           "LBP_AlarmMsgs".UserA[05].A70UUxx[00] := FALSE;

           "LBP_AlarmMsgs".UserA[06].A70UUxx[00] := FALSE;
           "LBP_AlarmMsgs".UserA[06].A70UUxx[01] := FALSE;
           "LBP_AlarmMsgs".UserA[06].A70UUxx[02] := FALSE;
           "LBP_AlarmMsgs".UserA[06].A70UUxx[03] := FALSE;
           "LBP_AlarmMsgs".UserA[06].A70UUxx[23] := FALSE;
           "LBP_AlarmMsgs".UserA[06].A70UUxx[25] := FALSE;
       END_IF;
   END_REGION

   REGION Ack alarm level 6
       IF "MCP1_In".reset THEN
           "LBP_AlarmMsgs".UserA[04].A70UUxx[02] := FALSE;
       END_IF;
   END_REGION

   REGION Ack alarm RID 5102xx
       IF "LBP_Chan1".E_ChanReset THEN
           "LBP_AlarmMsgs".ChanA[1].RID_5C02xx[00] := FALSE;
           "LBP_AlarmMsgs".ChanA[1].RID_5C02xx[01] := FALSE;
           "LBP_AlarmMsgs".ChanA[1].RID_5C02xx[02] := FALSE;
           "LBP_AlarmMsgs".ChanA[1].RID_5C02xx[03] := FALSE;
           "LBP_AlarmMsgs".ChanA[1].RID_5C02xx[04] := FALSE;
           "LBP_AlarmMsgs".ChanA[1].RID_5C02xx[05] := FALSE;
           "LBP_AlarmMsgs".ChanA[1].RID_5C02xx[06] := FALSE;
           "LBP_AlarmMsgs".ChanA[1].RID_5C02xx[07] := FALSE;
           "LBP_AlarmMsgs".ChanA[1].RID_5C02xx[08] := FALSE;
           "LBP_AlarmMsgs".ChanA[1].RID_5C02xx[09] := FALSE;
           "LBP_AlarmMsgs".ChanA[1].RID_5C02xx[10] := FALSE;
           "LBP_AlarmMsgs".ChanA[1].RID_5C02xx[11] := FALSE;
           "LBP_AlarmMsgs".ChanA[1].RID_5C02xx[12] := FALSE;
           "LBP_AlarmMsgs".ChanA[1].RID_5C02xx[13] := FALSE;
           "LBP_AlarmMsgs".ChanA[1].RID_5C02xx[14] := FALSE;
           "LBP_AlarmMsgs".ChanA[1].RID_5C02xx[15] := FALSE;
       END_IF;
   END_REGION
END_FUNCTION_BLOCK

FUNCTION_BLOCK "FB_Msg"   // FB84, SCL
{ S7_Optimized_Access := 'TRUE' }
// stored: MemoryReserve 100, SetENOAutomatically false
   VAR
      sSeverity : Byte;
      sMemoNumberOfActiveAlarms : DInt;
      sTON_On : TON_TIME;
      sTON_OFF { S7_SetPoint := 'True'} : TON_TIME;
      sPulseUpdateAlarms { S7_SetPoint := 'True'} : Bool;
      sRT_PulseUpdateAlarms : R_TRIG;
   END_VAR
   VAR_TEMP
      tIndex1 : Int;
      tIndex2 : Int;
      tResultByte0 : Int;
   END_VAR
   VAR CONSTANT
      MSG_SIZE : Int := 95;
   END_VAR
BEGIN
   // REGION Test
   //     FOR #tIndex := 0 TO #MSG_SIZE DO
   //         #tResultByte0 := PEEK(area := 16#84, dbNumber := 2, byteOffset := #tIndex + 554);
   //         "Db_Messages".Msg[#tIndex].ID := #tIndex;
   //         "Db_Messages".Msg[#tIndex].Number := INT_TO_DINT(#tIndex) + 70000;
   //         "Db_Messages".Msg[#tIndex].Active := #tResultByte0.%X0;
   //     END_FOR;
   // END_REGION

   REGION Format Msg
       // Mise en forme des alarmes (DB2) dans DB_FormatMsg
       FOR #tIndex1 := 0 TO 8 DO
           FOR #tIndex2 := 0 TO 7 DO
               #tResultByte0 := PEEK(area := 16#84, dbNumber := 2, byteOffset := #tIndex2 + 554 + (#tIndex1 * 8));
               "DB_FormatMsg".Msg[(#tIndex2 * 8) + (#tIndex1 * 64) + 0].Id := INT_TO_DINT((#tIndex2 * 8) + 0) + 70000 + (#tIndex1 * 100);
               "DB_FormatMsg".Msg[(#tIndex2 * 8) + (#tIndex1 * 64) + 1].Id := INT_TO_DINT((#tIndex2 * 8) + 1) + 70000 + (#tIndex1 * 100);
               "DB_FormatMsg".Msg[(#tIndex2 * 8) + (#tIndex1 * 64) + 2].Id := INT_TO_DINT((#tIndex2 * 8) + 2) + 70000 + (#tIndex1 * 100);
               "DB_FormatMsg".Msg[(#tIndex2 * 8) + (#tIndex1 * 64) + 3].Id := INT_TO_DINT((#tIndex2 * 8) + 3) + 70000 + (#tIndex1 * 100);
               "DB_FormatMsg".Msg[(#tIndex2 * 8) + (#tIndex1 * 64) + 4].Id := INT_TO_DINT((#tIndex2 * 8) + 4) + 70000 + (#tIndex1 * 100);
               "DB_FormatMsg".Msg[(#tIndex2 * 8) + (#tIndex1 * 64) + 5].Id := INT_TO_DINT((#tIndex2 * 8) + 5) + 70000 + (#tIndex1 * 100);
               "DB_FormatMsg".Msg[(#tIndex2 * 8) + (#tIndex1 * 64) + 6].Id := INT_TO_DINT((#tIndex2 * 8) + 6) + 70000 + (#tIndex1 * 100);
               "DB_FormatMsg".Msg[(#tIndex2 * 8) + (#tIndex1 * 64) + 7].Id := INT_TO_DINT((#tIndex2 * 8) + 7) + 70000 + (#tIndex1 * 100);

               "DB_FormatMsg".Msg[(#tIndex2 * 8) + (#tIndex1 * 64) + 0].Active := #tResultByte0.%X0;
               "DB_FormatMsg".Msg[(#tIndex2 * 8) + (#tIndex1 * 64) + 1].Active := #tResultByte0.%X1;
               "DB_FormatMsg".Msg[(#tIndex2 * 8) + (#tIndex1 * 64) + 2].Active := #tResultByte0.%X2;
               "DB_FormatMsg".Msg[(#tIndex2 * 8) + (#tIndex1 * 64) + 3].Active := #tResultByte0.%X3;
               "DB_FormatMsg".Msg[(#tIndex2 * 8) + (#tIndex1 * 64) + 4].Active := #tResultByte0.%X4;
               "DB_FormatMsg".Msg[(#tIndex2 * 8) + (#tIndex1 * 64) + 5].Active := #tResultByte0.%X5;
               "DB_FormatMsg".Msg[(#tIndex2 * 8) + (#tIndex1 * 64) + 6].Active := #tResultByte0.%X6;
               "DB_FormatMsg".Msg[(#tIndex2 * 8) + (#tIndex1 * 64) + 7].Active := #tResultByte0.%X7;
           END_FOR;
       END_FOR;
   END_REGION

   REGION Severity WFA A REVOIR !!
       #sSeverity := 1;
       "DB_FormatMsg".Msg[35].Severity := #sSeverity;

       "DB_FormatMsg".Msg[236].Severity := #sSeverity;

       "DB_FormatMsg".Msg[532].Severity := #sSeverity;
       "DB_FormatMsg".Msg[533].Severity := #sSeverity;
       "DB_FormatMsg".Msg[534].Severity := #sSeverity;
       "DB_FormatMsg".Msg[535].Severity := #sSeverity;
       "DB_FormatMsg".Msg[536].Severity := #sSeverity;
       "DB_FormatMsg".Msg[537].Severity := #sSeverity;
       "DB_FormatMsg".Msg[538].Severity := #sSeverity;
       "DB_FormatMsg".Msg[539].Severity := #sSeverity;
       "DB_FormatMsg".Msg[542].Severity := #sSeverity;
       "DB_FormatMsg".Msg[548].Severity := #sSeverity;
       "DB_FormatMsg".Msg[550].Severity := #sSeverity;
       "DB_FormatMsg".Msg[551].Severity := #sSeverity;

       "DB_FormatMsg".Msg[800].Severity := #sSeverity;
       "DB_FormatMsg".Msg[841].Severity := #sSeverity;

       #sSeverity := 2;
       "DB_FormatMsg".Msg[59].Severity := #sSeverity;
       "DB_FormatMsg".Msg[60].Severity := #sSeverity;
       "DB_FormatMsg".Msg[61].Severity := #sSeverity;
       "DB_FormatMsg".Msg[62].Severity := #sSeverity;

       "DB_FormatMsg".Msg[348].Severity := #sSeverity;

       "DB_FormatMsg".Msg[441].Severity := #sSeverity;
       "DB_FormatMsg".Msg[442].Severity := #sSeverity;

       "DB_FormatMsg".Msg[543].Severity := #sSeverity;

       "DB_FormatMsg".Msg[662].Severity := #sSeverity;
       "DB_FormatMsg".Msg[663].Severity := #sSeverity;

       // "DB_FormatMsg".Msg[3032].Severity := #sSeverity;
       // "DB_FormatMsg".Msg[3033].Severity := #sSeverity;
       // "DB_FormatMsg".Msg[3034].Severity := #sSeverity;
       // "DB_FormatMsg".Msg[3035].Severity := #sSeverity;
       // "DB_FormatMsg".Msg[3036].Severity := #sSeverity;
       // "DB_FormatMsg".Msg[3037].Severity := #sSeverity;
       // "DB_FormatMsg".Msg[3038].Severity := #sSeverity;
       // "DB_FormatMsg".Msg[3039].Severity := #sSeverity;
       // "DB_FormatMsg".Msg[3010].Severity := #sSeverity;
       // "DB_FormatMsg".Msg[3041].Severity := #sSeverity;
       // "DB_FormatMsg".Msg[3042].Severity := #sSeverity;
       // "DB_FormatMsg".Msg[3043].Severity := #sSeverity;
       // "DB_FormatMsg".Msg[3044].Severity := #sSeverity;
       // "DB_FormatMsg".Msg[3045].Severity := #sSeverity;
       // "DB_FormatMsg".Msg[3046].Severity := #sSeverity;
       // "DB_FormatMsg".Msg[3047].Severity := #sSeverity;


       "DB_FormatMsg".Msg[55].Severity := #sSeverity;
       "DB_FormatMsg".Msg[63].Severity := #sSeverity;

       "DB_FormatMsg".Msg[403].Severity := #sSeverity;
       "DB_FormatMsg".Msg[404].Severity := #sSeverity;
       "DB_FormatMsg".Msg[405].Severity := #sSeverity;
       "DB_FormatMsg".Msg[406].Severity := #sSeverity;
       "DB_FormatMsg".Msg[420].Severity := #sSeverity;
       "DB_FormatMsg".Msg[421].Severity := #sSeverity;
       "DB_FormatMsg".Msg[422].Severity := #sSeverity;
       "DB_FormatMsg".Msg[423].Severity := #sSeverity;

       "DB_FormatMsg".Msg[508].Severity := #sSeverity;
       "DB_FormatMsg".Msg[509].Severity := #sSeverity;
       "DB_FormatMsg".Msg[510].Severity := #sSeverity;
       "DB_FormatMsg".Msg[511].Severity := #sSeverity;
       "DB_FormatMsg".Msg[512].Severity := #sSeverity;

       "DB_FormatMsg".Msg[652].Severity := #sSeverity;
       "DB_FormatMsg".Msg[653].Severity := #sSeverity;

       "DB_FormatMsg".Msg[700].Severity := #sSeverity;
       "DB_FormatMsg".Msg[701].Severity := #sSeverity;
       "DB_FormatMsg".Msg[702].Severity := #sSeverity;
       "DB_FormatMsg".Msg[703].Severity := #sSeverity;
       "DB_FormatMsg".Msg[704].Severity := #sSeverity;
       "DB_FormatMsg".Msg[705].Severity := #sSeverity;
       "DB_FormatMsg".Msg[706].Severity := #sSeverity;
       "DB_FormatMsg".Msg[707].Severity := #sSeverity;
       "DB_FormatMsg".Msg[708].Severity := #sSeverity;
       "DB_FormatMsg".Msg[709].Severity := #sSeverity;
       "DB_FormatMsg".Msg[710].Severity := #sSeverity;
       "DB_FormatMsg".Msg[711].Severity := #sSeverity;
       "DB_FormatMsg".Msg[740].Severity := #sSeverity;
       "DB_FormatMsg".Msg[741].Severity := #sSeverity;
       "DB_FormatMsg".Msg[742].Severity := #sSeverity;
       "DB_FormatMsg".Msg[743].Severity := #sSeverity;
       "DB_FormatMsg".Msg[744].Severity := #sSeverity;
       "DB_FormatMsg".Msg[745].Severity := #sSeverity;
       "DB_FormatMsg".Msg[746].Severity := #sSeverity;
       "DB_FormatMsg".Msg[747].Severity := #sSeverity;
       "DB_FormatMsg".Msg[748].Severity := #sSeverity;
       "DB_FormatMsg".Msg[749].Severity := #sSeverity;
       "DB_FormatMsg".Msg[750].Severity := #sSeverity;
       "DB_FormatMsg".Msg[751].Severity := #sSeverity;
       "DB_FormatMsg".Msg[752].Severity := #sSeverity;
       "DB_FormatMsg".Msg[753].Severity := #sSeverity;
       "DB_FormatMsg".Msg[754].Severity := #sSeverity;
       "DB_FormatMsg".Msg[755].Severity := #sSeverity;
       "DB_FormatMsg".Msg[756].Severity := #sSeverity;
       "DB_FormatMsg".Msg[757].Severity := #sSeverity;
       "DB_FormatMsg".Msg[758].Severity := #sSeverity;
       "DB_FormatMsg".Msg[759].Severity := #sSeverity;
       "DB_FormatMsg".Msg[760].Severity := #sSeverity;
       "DB_FormatMsg".Msg[761].Severity := #sSeverity;

       // "DB_FormatMsg".Msg[3000].Severity := #sSeverity;
       // "DB_FormatMsg".Msg[3001].Severity := #sSeverity;
       // "DB_FormatMsg".Msg[3002].Severity := #sSeverity;
       // "DB_FormatMsg".Msg[3003].Severity := #sSeverity;
       // "DB_FormatMsg".Msg[3004].Severity := #sSeverity;
       // "DB_FormatMsg".Msg[3005].Severity := #sSeverity;
       // "DB_FormatMsg".Msg[3006].Severity := #sSeverity;
       // "DB_FormatMsg".Msg[3007].Severity := #sSeverity;
       // "DB_FormatMsg".Msg[3008].Severity := #sSeverity;
       // "DB_FormatMsg".Msg[3009].Severity := #sSeverity;
       // "DB_FormatMsg".Msg[3010].Severity := #sSeverity;
       // "DB_FormatMsg".Msg[3011].Severity := #sSeverity;
       // "DB_FormatMsg".Msg[3012].Severity := #sSeverity;
       // "DB_FormatMsg".Msg[3013].Severity := #sSeverity;
       // "DB_FormatMsg".Msg[3014].Severity := #sSeverity;
       // "DB_FormatMsg".Msg[3015].Severity := #sSeverity;


       #sSeverity := 3;
       "DB_FormatMsg".Msg[6].Severity := #sSeverity;
       "DB_FormatMsg".Msg[7].Severity := #sSeverity;
       "DB_FormatMsg".Msg[8].Severity := #sSeverity;

       "DB_FormatMsg".Msg[103].Severity := #sSeverity;
       "DB_FormatMsg".Msg[104].Severity := #sSeverity;
       "DB_FormatMsg".Msg[105].Severity := #sSeverity;
       "DB_FormatMsg".Msg[106].Severity := #sSeverity;
       "DB_FormatMsg".Msg[107].Severity := #sSeverity;
       "DB_FormatMsg".Msg[108].Severity := #sSeverity;
       "DB_FormatMsg".Msg[109].Severity := #sSeverity;
       "DB_FormatMsg".Msg[110].Severity := #sSeverity;
       "DB_FormatMsg".Msg[111].Severity := #sSeverity;
       "DB_FormatMsg".Msg[112].Severity := #sSeverity;
       "DB_FormatMsg".Msg[113].Severity := #sSeverity;
       "DB_FormatMsg".Msg[114].Severity := #sSeverity;
       "DB_FormatMsg".Msg[115].Severity := #sSeverity;
       "DB_FormatMsg".Msg[120].Severity := #sSeverity;

       "DB_FormatMsg".Msg[200].Severity := #sSeverity;
       "DB_FormatMsg".Msg[201].Severity := #sSeverity;
       "DB_FormatMsg".Msg[202].Severity := #sSeverity;
       "DB_FormatMsg".Msg[204].Severity := #sSeverity;
       "DB_FormatMsg".Msg[205].Severity := #sSeverity;
       "DB_FormatMsg".Msg[206].Severity := #sSeverity;
       "DB_FormatMsg".Msg[207].Severity := #sSeverity;
       "DB_FormatMsg".Msg[208].Severity := #sSeverity;
       "DB_FormatMsg".Msg[209].Severity := #sSeverity;
       "DB_FormatMsg".Msg[210].Severity := #sSeverity;
       "DB_FormatMsg".Msg[211].Severity := #sSeverity;
       "DB_FormatMsg".Msg[212].Severity := #sSeverity;
       "DB_FormatMsg".Msg[218].Severity := #sSeverity;
       "DB_FormatMsg".Msg[219].Severity := #sSeverity;
       "DB_FormatMsg".Msg[220].Severity := #sSeverity;
       "DB_FormatMsg".Msg[221].Severity := #sSeverity;
       "DB_FormatMsg".Msg[222].Severity := #sSeverity;

       "DB_FormatMsg".Msg[315].Severity := #sSeverity;
       "DB_FormatMsg".Msg[316].Severity := #sSeverity;
       "DB_FormatMsg".Msg[317].Severity := #sSeverity;
       "DB_FormatMsg".Msg[318].Severity := #sSeverity;
       "DB_FormatMsg".Msg[319].Severity := #sSeverity;
       "DB_FormatMsg".Msg[320].Severity := #sSeverity;
       "DB_FormatMsg".Msg[321].Severity := #sSeverity;
       "DB_FormatMsg".Msg[322].Severity := #sSeverity;
       "DB_FormatMsg".Msg[323].Severity := #sSeverity;
       "DB_FormatMsg".Msg[324].Severity := #sSeverity;
       "DB_FormatMsg".Msg[325].Severity := #sSeverity;
       "DB_FormatMsg".Msg[326].Severity := #sSeverity;

       "DB_FormatMsg".Msg[409].Severity := #sSeverity;
       "DB_FormatMsg".Msg[410].Severity := #sSeverity;
       "DB_FormatMsg".Msg[424].Severity := #sSeverity;
       "DB_FormatMsg".Msg[425].Severity := #sSeverity;
       "DB_FormatMsg".Msg[426].Severity := #sSeverity;
       "DB_FormatMsg".Msg[427].Severity := #sSeverity;
       "DB_FormatMsg".Msg[428].Severity := #sSeverity;
       "DB_FormatMsg".Msg[429].Severity := #sSeverity;

       "DB_FormatMsg".Msg[604].Severity := #sSeverity;
       "DB_FormatMsg".Msg[605].Severity := #sSeverity;
       "DB_FormatMsg".Msg[606].Severity := #sSeverity;
       "DB_FormatMsg".Msg[607].Severity := #sSeverity;
       "DB_FormatMsg".Msg[608].Severity := #sSeverity;
       "DB_FormatMsg".Msg[609].Severity := #sSeverity;
       "DB_FormatMsg".Msg[610].Severity := #sSeverity;
       "DB_FormatMsg".Msg[611].Severity := #sSeverity;
       "DB_FormatMsg".Msg[640].Severity := #sSeverity;
       "DB_FormatMsg".Msg[641].Severity := #sSeverity;
       "DB_FormatMsg".Msg[650].Severity := #sSeverity;
       "DB_FormatMsg".Msg[651].Severity := #sSeverity;
       "DB_FormatMsg".Msg[654].Severity := #sSeverity;
       "DB_FormatMsg".Msg[655].Severity := #sSeverity;
       "DB_FormatMsg".Msg[656].Severity := #sSeverity;
       "DB_FormatMsg".Msg[657].Severity := #sSeverity;
       "DB_FormatMsg".Msg[658].Severity := #sSeverity;
       "DB_FormatMsg".Msg[659].Severity := #sSeverity;
       "DB_FormatMsg".Msg[660].Severity := #sSeverity;
       "DB_FormatMsg".Msg[661].Severity := #sSeverity;

       "DB_FormatMsg".Msg[808].Severity := #sSeverity;
       "DB_FormatMsg".Msg[809].Severity := #sSeverity;
       "DB_FormatMsg".Msg[810].Severity := #sSeverity;
       "DB_FormatMsg".Msg[811].Severity := #sSeverity;
       "DB_FormatMsg".Msg[812].Severity := #sSeverity;
       "DB_FormatMsg".Msg[813].Severity := #sSeverity;
       "DB_FormatMsg".Msg[814].Severity := #sSeverity;
       "DB_FormatMsg".Msg[815].Severity := #sSeverity;
       "DB_FormatMsg".Msg[816].Severity := #sSeverity;
       "DB_FormatMsg".Msg[817].Severity := #sSeverity;
       "DB_FormatMsg".Msg[820].Severity := #sSeverity;
       "DB_FormatMsg".Msg[821].Severity := #sSeverity;
       "DB_FormatMsg".Msg[822].Severity := #sSeverity;
       "DB_FormatMsg".Msg[823].Severity := #sSeverity;
       "DB_FormatMsg".Msg[824].Severity := #sSeverity;

       "DB_FormatMsg".Msg[2].Severity := #sSeverity;
       "DB_FormatMsg".Msg[5].Severity := #sSeverity;

       "DB_FormatMsg".Msg[501].Severity := #sSeverity;
       "DB_FormatMsg".Msg[502].Severity := #sSeverity;

       "DB_FormatMsg".Msg[642].Severity := #sSeverity;
       "DB_FormatMsg".Msg[643].Severity := #sSeverity;
       "DB_FormatMsg".Msg[644].Severity := #sSeverity;
       "DB_FormatMsg".Msg[645].Severity := #sSeverity;
       "DB_FormatMsg".Msg[646].Severity := #sSeverity;
       "DB_FormatMsg".Msg[647].Severity := #sSeverity;
       "DB_FormatMsg".Msg[648].Severity := #sSeverity;
       "DB_FormatMsg".Msg[649].Severity := #sSeverity;

       #sSeverity := 4;
       "DB_FormatMsg".Msg[3].Severity := #sSeverity;
       "DB_FormatMsg".Msg[4].Severity := #sSeverity;

       "DB_FormatMsg".Msg[330].Severity := #sSeverity;
       "DB_FormatMsg".Msg[331].Severity := #sSeverity;

       "DB_FormatMsg".Msg[500].Severity := #sSeverity;

       "DB_FormatMsg".Msg[600].Severity := #sSeverity;
       "DB_FormatMsg".Msg[601].Severity := #sSeverity;
       "DB_FormatMsg".Msg[602].Severity := #sSeverity;
       "DB_FormatMsg".Msg[603].Severity := #sSeverity;
       "DB_FormatMsg".Msg[623].Severity := #sSeverity;
       "DB_FormatMsg".Msg[625].Severity := #sSeverity;

       "DB_FormatMsg".Msg[402].Severity := #sSeverity;
   END_REGION

   REGION Active Alarms
       // Recherche des alarmes actives dans DB_FormatMsg
       #tIndex2 := 0;
       FOR #tIndex1 := 0 TO 575 DO
           IF "DB_FormatMsg".Msg[#tIndex1].Active THEN
               "DB_ActiveAlarms".ActiveAlarms[#tIndex2].Id := "DB_FormatMsg".Msg[#tIndex1].Id;
               "DB_ActiveAlarms".ActiveAlarms[#tIndex2].Severity := "DB_FormatMsg".Msg[#tIndex1].Severity;
               #tIndex2 := #tIndex2 + 1;
           END_IF;
       END_FOR;
       "DB_ActiveAlarms".NumberOfActiveAlarms := #tIndex2;
   END_REGION

   REGION Update alarms
       // TON phase ON (5 secondes)
       #sTON_On(
                IN := #sPulseUpdateAlarms,
                PT := T#5s);

       // TON phase OFF (5 secondes)
       #sTON_OFF(
                 IN := NOT #sPulseUpdateAlarms,
                 PT := T#5s);

       IF #sTON_On.Q THEN
           #sPulseUpdateAlarms := FALSE;
       END_IF;

       IF #sTON_OFF.Q THEN
           #sPulseUpdateAlarms := TRUE;
       END_IF;

       #sRT_PulseUpdateAlarms(CLK := #sPulseUpdateAlarms);

       IF ("DB_ActiveAlarms".NumberOfActiveAlarms <> #sMemoNumberOfActiveAlarms) OR #sRT_PulseUpdateAlarms.Q THEN
           "DB_ActiveAlarms".Update := "DB_ActiveAlarms".Update + 1;
           IF "DB_ActiveAlarms".Update > 255 OR "DB_ActiveAlarms".Update < 1 THEN
               "DB_ActiveAlarms".Update := 1;
           END_IF;
       END_IF;
   END_REGION

   REGION Transfert to OPC
       "DB_OPC_Alarms".ActiveAlarms := "DB_ActiveAlarms".ActiveAlarms;
       "DB_OPC_Alarms".NumberOfActiveAlarms := "DB_ActiveAlarms".NumberOfActiveAlarms;
       "DB_OPC_Alarms".Update := "DB_ActiveAlarms".Update;
   END_REGION
END_FUNCTION_BLOCK

FUNCTION_BLOCK "FB_DecodChannels"   // FB405, SCL
{ S7_Optimized_Access := 'TRUE' }
// stored: AutoNumber false, MemoryReserve 100, SetENOAutomatically false
   VAR DB_SPECIFIC
      sChan1IsDisplayed : Bool;
      sChan2IsDisplayed : Bool;
      sChan3IsDisplayed : Bool;
      sChan4IsDisplayed : Bool;
   END_VAR
   VAR CONSTANT
      CH00 : Byte := 0;
      CH01 : Byte := 1;
      CH02 : Byte := 2;
      CH03 : Byte := 3;
      CH04 : Byte := 4;
   END_VAR
BEGIN
   REGION Description header 
       //==================================================================================
       // POSALUX Swiss SA / (C) Copyright 2025
       //----------------------------------------------------------------------------------
       // Title: FB_DecodChannels
       // Comment/Function: Indication of the displayed channel according to the
       //                   current channel number
       // Author: Fabien WALDT
       // Engineering: TIA Portal v17
       //----------------------------------------------------------------------------------
       // Change log table:
       // Version  | Date     | Expert in charge | Changes applied
       // ---------|----------|------------------|-----------------------------------------
       // 00.00.01 | 20250505 | WFA              | First released version
       // =================================================================================
   END_REGION

   REGION Channel decoding
       CASE "LBP_HMI".E_Chan OF
           #CH00:
               #sChan1IsDisplayed := 0;
               #sChan2IsDisplayed := 0;
               #sChan3IsDisplayed := 0;
               #sChan4IsDisplayed := 0;
           #CH01:
               #sChan1IsDisplayed := 1;
               #sChan2IsDisplayed := 0;
               #sChan3IsDisplayed := 0;
               #sChan4IsDisplayed := 0;
           #CH02:
               #sChan1IsDisplayed := 0;
               #sChan2IsDisplayed := 1;
               #sChan3IsDisplayed := 0;
               #sChan4IsDisplayed := 0;
           #CH03:
               #sChan1IsDisplayed := 0;
               #sChan2IsDisplayed := 0;
               #sChan3IsDisplayed := 1;
               #sChan4IsDisplayed := 0;
           #CH04:
               #sChan1IsDisplayed := 0;
               #sChan2IsDisplayed := 0;
               #sChan3IsDisplayed := 0;
               #sChan4IsDisplayed := 1;
           ELSE
               #sChan1IsDisplayed := 0;
               #sChan2IsDisplayed := 0;
               #sChan3IsDisplayed := 0;
               #sChan4IsDisplayed := 0;
       END_CASE;
   END_REGION
END_FUNCTION_BLOCK

FUNCTION_BLOCK "FB_CycleStartStop"   // FB406, SCL
{ S7_Optimized_Access := 'TRUE' }
// stored: AutoNumber false, MemoryReserve 100, SetENOAutomatically false
   VAR
      sChan1Start : Bool;
      sResquestStopNextCycle : Bool;
      sTimePowerSupplyAlarm : TON_TIME;
      sRT_CNAskStopCycle : R_TRIG;
   END_VAR
   VAR CONSTANT
      TIME_POWER_SUPPPLY_ALARM : Time := T#5s;
   END_VAR
BEGIN
   REGION Description header 
       //==================================================================================
       // POSALUX Swiss SA / (C) Copyright 2024
       //----------------------------------------------------------------------------------
       // Title: Start and stop cycle
       // Comment/Function:  Replacement of the Siemens standard cycle stop button with a
       // customized method for stopping and restarting the cycle, adabted to the specific
       // needs of the application.
       // 
       // Author: Gowsigan SRITHARAN
       // Engineering: TIA Portal v17
       //----------------------------------------------------------------------------------
       // Change log table:
       // Version  | Date     | Expert in charge | Changes applied
       // ---------|----------|------------------|------------------------------------
       // 00.00.01 | 20241202 | GSR              | First released version
       // ==================================================================================
   END_REGION

   REGION Start memo
       // Start channel
       IF "LBP_Chan1".E_ProgRunning THEN
           #sChan1Start := TRUE;
       END_IF;

       // Reset channel
       IF "LBP_Chan1".E_ChanReset THEN
           #sChan1Start := FALSE;
       END_IF;
   END_REGION

   REGION Start disabled
       "LBP_Chan1".A_NCStartDisabl :="DB_Alarms".sAlarmsLevel3 OR "DB_Alarms".sAlarmsLevel4 OR "DB_Alarms".sAlarmsLevel5 OR  "DB_Alarms".sAlarmsLevel6;
       "LBP_Chan1".A_NCStart := ("MCP1_In".cycleStart OR "DB_HMISetting".StartAutoReq) AND (NOT"LBP_Chan1".A_NCStartDisabl);

       "DB_HMISetting".StartAutoReq := FALSE;
   END_REGION

   REGION Mode change disabled
       "LBP_ModeGroup".A_MCDisable := #sChan1Start AND NOT "LBP_Chan1".E_M01;    // Disable change CNC mode
   END_REGION

   REGION  Stop request (From MCP or alarms)
       // If key stop cycle is pressed or alarm level3 then request stop
       IF #sChan1Start
           AND (NOT "MCP1_In".cycleStop OR "DB_HMISetting".StopAutoReq OR "DB_Alarms".sAlarmsLevel3 OR "DB_Alarms".sAlarmsLevel4) THEN
           #sResquestStopNextCycle := TRUE;
           "LBP_AlarmMsgs".UserA[00].A70UUxx[60] := TRUE; // Msg "Stop program requested by operator"

           "DB_HMISetting".StopAutoReq := FALSE;
       END_IF;
   END_REGION

   REGION Wait Channel stopped
       IF  #sResquestStopNextCycle AND "LBP_Chan1".E_M01 THEN
           #sResquestStopNextCycle := FALSE;
       END_IF;
   END_REGION

   REGION Reset stop at next step
       IF "LBP_Chan1".MDyn[78] OR "LBP_Chan1".E_ChanReset THEN // M78 ISO command to restart 
           "LBP_NC".A_Set_Inp31 := FALSE;
           "LBP_AlarmMsgs".UserA[0].A70UUxx[60] := FALSE;
           #sResquestStopNextCycle := FALSE;
       END_IF;
   END_REGION

   REGION LED NC Start / Stop
       // Stop LED
       "MCP1_Out".LEDcycleStop :=
       NOT "LBP_Chan1".E_ChanReset
       AND NOT "LBP_Chan1".A_Ref
       AND ("LBP_Chan1".E_ProgStop
       OR "LBP_Chan1".E_ProgInterrupt
       OR "LBP_Chan1".E_ProgAborted) OR
       (#sResquestStopNextCycle AND "Clock_1Hz");

       // Start LED
       "MCP1_Out".LEDcycleStart :="LBP_Chan1".E_ProgRunning OR "LBP_Chan1".A_Ref;

      // Cycle start LED (Key [19])
       "DB_McpKeyboardSignals".sStartCycle.sLedSWStatus := "LBP_Chan1".E_ProgRunning OR "LBP_Chan1".A_Ref;
   END_REGION

   REGION Channel feed disable (Power Supply error)
       #sTimePowerSupplyAlarm(IN := "DB_PowerOn".sMachinePower
                              AND (NOT "DB_DigitalInputs".sPowerReady.sSWStatus
                              OR NOT "DB_DigitalInputs".sAlarmI2T.sSWStatus),
                              PT := #TIME_POWER_SUPPPLY_ALARM);

       IF #sTimePowerSupplyAlarm.Q THEN
           "LBP_AlarmMsgs".Chan[1].FDD[1] := TRUE;
       ELSIF "DB_McpKeyboardSignals".sAlarmReset.sKeySWStatus THEN
           "LBP_AlarmMsgs".Chan[1].FDD[1] := FALSE;
       END_IF;

       IF #sTimePowerSupplyAlarm.Q AND NOT "DB_DigitalInputs".sPowerReady.sSWStatus THEN
           "LBP_AlarmMsgs".UserA[03].A70UUxx[30] := TRUE;       // Msg: 700330 "Drives power supply not ready"
       END_IF;

       IF #sTimePowerSupplyAlarm.Q AND NOT "DB_DigitalInputs".sAlarmI2T.sSWStatus THEN
           "LBP_AlarmMsgs".UserA[03].A70UUxx[31] := TRUE;       // Msg: 700331 "Drives power supply overload"
       END_IF;
   END_REGION
END_FUNCTION_BLOCK

FUNCTION_BLOCK "FB_Axis"   // FB410, SCL
{ S7_Optimized_Access := 'TRUE' }
// stored: AutoNumber false, MemoryReserve 100, SetENOAutomatically false
   VAR
      "sBrakeTest ZM" { S7_SetPoint := 'True'} : "FB_BrakeTest";
      "sBrakeTest ZL" { S7_SetPoint := 'True'} : "FB_BrakeTest";
      "BrakeTest ZM" : Struct
         sSBTDone { S7_SetPoint := 'True'} : Bool;
         sStartSBT { S7_SetPoint := 'True'} : Bool;
         sDone { S7_SetPoint := 'True'} : Bool;
         sError : Bool;
         sStateNum : Int;
         sDiagnoseError : Int;
         scloseExternalBrake : Bool;
      END_STRUCT;
      "BrakeTest ZL" : Struct
         sSBTDone { S7_SetPoint := 'True'} : Bool;
         sStartSBT { S7_SetPoint := 'True'} : Bool;
         sDone { S7_SetPoint := 'True'} : Bool;
         sError : Bool;
         sStateNum : Int;
         sDiagnoseError : Int;
         scloseExternalBrake : Bool;
      END_STRUCT;
      sErrorN : Array[1..8] of Bool;
      sTestStopRequested : Bool;
      sTestStopStart : Bool;
      sTestStopError : Bool;
      sTestStopEnd : Bool;
      sTestStopDone : Bool;
      sLedSITestOK : Bool;
      sLedSITestSlowFlashing : Bool;
      sLedSITestQuickFlashing : Bool;
      sTimerTestStopStart : TON_TIME;
      sTimerTestStopEnd : TON_TIME;
   END_VAR
   VAR RETAIN
      DisableAxis01_X { S7_SetPoint := 'True'} : Bool;
      DisableAxis02_Y { S7_SetPoint := 'True'} : Bool;
      DisableAxis03_ZM { S7_SetPoint := 'True'} : Bool;
      DisableAxis04_B { S7_SetPoint := 'True'} : Bool;
      DisableAxis05_U1 { S7_SetPoint := 'True'} : Bool;
      DisableAxis06_U2 { S7_SetPoint := 'True'} : Bool;
      DisableAxis07_V { S7_SetPoint := 'True'} : Bool;
      DisableAxis08_W { S7_SetPoint := 'True'} : Bool;
      DisableAxis09_ZL { S7_SetPoint := 'True'} : Bool;
   END_VAR
BEGIN
   REGION Description header 
       //==================================================================================
       // POSALUX Swiss SA / (C) Copyright 2025
       //----------------------------------------------------------------------------------
       // Title: FB_Axis
       // Comment/Function: 
       // Author: Fabien WALDT
       // Engineering: TIA Portal v17
       //----------------------------------------------------------------------------------
       // Change log table:
       // Version  | Date     | Expert in charge | Changes applied
       // ---------|----------|------------------|-----------------------------------------
       // 00.00.01 | 20250423 | WFA              | First released version
       // =================================================================================
   END_REGION

   REGION Axis disable
       "LBP_Axis01_X".A_ASpDisable  := FALSE;
       "LBP_Axis02_Y".A_ASpDisable  := FALSE;
       "LBP_Axis03_ZM".A_ASpDisable := FALSE;
       "LBP_Axis04_B".A_ASpDisable  := FALSE;
       "LBP_Axis05_U1".A_ASpDisable := FALSE;
       "LBP_Axis06_U2".A_ASpDisable := FALSE;
       "LBP_Axis07_V".A_ASpDisable  := FALSE;
       "LBP_Axis08_W".A_ASpDisable  := FALSE;
       "LBP_Axis09_ZL".A_ASpDisable := FALSE;
   END_REGION

   REGION Axis follow-up mode
       "LBP_Axis01_X".A_Follow_upMode  := TRUE;
       "LBP_Axis02_Y".A_Follow_upMode  := TRUE;
       "LBP_Axis03_ZM".A_Follow_upMode := TRUE;
       "LBP_Axis04_B".A_Follow_upMode  := TRUE;
       "LBP_Axis05_U1".A_Follow_upMode := TRUE;
       "LBP_Axis06_U2".A_Follow_upMode := TRUE;
       "LBP_Axis07_V".A_Follow_upMode  := TRUE;
       "LBP_Axis08_W".A_Follow_upMode  := TRUE;
       "LBP_Axis09_ZL".A_Follow_upMode := TRUE;
   END_REGION

   REGION Measure system selection
       "LBP_Axis01_X".A_PosMeas1  := TRUE;
       "LBP_Axis01_X".A_PosMeas2  := FALSE;
       "LBP_Axis02_Y".A_PosMeas1  := TRUE;
       "LBP_Axis02_Y".A_PosMeas2  := FALSE;
       "LBP_Axis03_ZM".A_PosMeas1 := FALSE;
       "LBP_Axis03_ZM".A_PosMeas2 := TRUE;
       "LBP_Axis04_B".A_PosMeas1  := TRUE;
       "LBP_Axis04_B".A_PosMeas2  := FALSE;
       "LBP_Axis05_U1".A_PosMeas1 := TRUE;
       "LBP_Axis05_U1".A_PosMeas2 := FALSE;
       "LBP_Axis06_U2".A_PosMeas1 := TRUE;
       "LBP_Axis06_U2".A_PosMeas2 := FALSE;
       "LBP_Axis07_V".A_PosMeas1  := TRUE;
       "LBP_Axis07_V".A_PosMeas2  := FALSE;
       "LBP_Axis08_W".A_PosMeas1  := TRUE;
       "LBP_Axis08_W".A_PosMeas2  := FALSE;
       "LBP_Axis09_ZL".A_PosMeas1 := FALSE;
       "LBP_Axis09_ZL".A_PosMeas2 := TRUE;
   END_REGION

   REGION Controle enable
       "LBP_Axis01_X".A_ContrEnable  := NOT #DisableAxis01_X;
       "LBP_Axis02_Y".A_ContrEnable  := NOT #DisableAxis02_Y;
       "LBP_Axis03_ZM".A_ContrEnable := NOT #DisableAxis03_ZM;
       "LBP_Axis04_B".A_ContrEnable  := NOT #DisableAxis04_B;
       "LBP_Axis05_U1".A_ContrEnable := NOT #DisableAxis05_U1;
       "LBP_Axis06_U2".A_ContrEnable := NOT #DisableAxis06_U2;
       "LBP_Axis07_V".A_ContrEnable  := NOT #DisableAxis07_V;
       "LBP_Axis08_W".A_ContrEnable  := NOT #DisableAxis08_W;
       "LBP_Axis09_ZL".A_ContrEnable := NOT #DisableAxis09_ZL;
   END_REGION

   REGION Pulse enable
       "LBP_Axis01_X".A_PulseEnable  := NOT #DisableAxis01_X;
       "LBP_Axis02_Y".A_PulseEnable  := NOT #DisableAxis02_Y;
       "LBP_Axis03_ZM".A_PulseEnable := NOT #DisableAxis03_ZM;
       "LBP_Axis04_B".A_PulseEnable  := NOT #DisableAxis04_B;
       "LBP_Axis05_U1".A_PulseEnable := NOT #DisableAxis05_U1;
       "LBP_Axis06_U2".A_PulseEnable := NOT #DisableAxis06_U2;
       "LBP_Axis07_V".A_PulseEnable  := NOT #DisableAxis07_V;
       "LBP_Axis08_W".A_PulseEnable  := NOT #DisableAxis08_W;
       "LBP_Axis09_ZL".A_PulseEnable := NOT #DisableAxis09_ZL;
   END_REGION

   REGION Axis04 B - Delay reference point approach
       "LBP_Axis04_B".A_DelayRef :="DB_DigitalInputs".sB_AxisReferencePoint.sSWStatus;
   END_REGION

   REGION Axis04 B - Feed Stop
       "LBP_Axis04_B".A_FDSpStop := (NOT "DB_DigitalOutputs".sClampingClosing.sSWStatus OR "DB_DigitalInputs".sClampingOpenCtrl.sSWStatus)
       OR "DB_AxisPosition".sAxis01_X."$AA_IM" < 95.0; // B Rotation diseable when X Axis is in laser area
   END_REGION

   REGION Axis05 U1 - Feed Stop
       "LBP_Axis05_U1".A_FDSpStop :=
       ("DB_LoaderShuttle1".sShuttlePosExt AND "DB_LoaderAxis".iU1PosSetPoint > "DB_AxisPosMachinePLC".Axis_U1.ExtGateExt AND NOT "DB_DigitalInputs".sExternalGateOpened.sSWStatus)       // Shuttle EXT - Consigne SAS/INT - Sas EXT pas ouvert
        OR ("DB_LoaderShuttle1".sShuttlePosSas AND "DB_LoaderAxis".iU1PosSetPoint < "DB_AxisPosMachinePLC".Axis_U1.IntGateExt AND NOT "DB_DigitalInputs".sExternalGateOpened.sSWStatus)    // Shuttle SAS - Consigne EXT     - Sas EXT pas ouvert
        OR ("DB_LoaderShuttle1".sShuttlePosSas AND "DB_LoaderAxis".iU1PosSetPoint > "DB_AxisPosMachinePLC".Axis_U1.ExtGateInt AND NOT "DB_DigitalInputs".sInternalGateOpened.sSWStatus)    // Shuttle SAS - Consigne INT     - Sas INT pas ouvert
        OR ("DB_LoaderShuttle1".sShuttlePosInt AND "DB_LoaderAxis".iU1PosSetPoint < "DB_AxisPosMachinePLC".Axis_U1.IntGateInt AND NOT "DB_DigitalInputs".sInternalGateOpened.sSWStatus)    // Shuttle INT - Consigne SAS/EXT - Sas INT pas ouvert
        OR ("DB_LoaderShuttle1".sShuttlePosInt AND NOT "DB_LoaderShuttle1".sIntLoaderInSafePos)                                                                                            // Shuttle INT - Int loader in safe position
        OR ("DB_LoaderShuttle1".sShuttlePosExt AND NOT "DB_LoaderShuttle1".sBwLoaderInSafePos) 
        OR ("DB_LoaderShuttle1".sShuttlePosExt AND "DB_BwLoader".sBwCommunication.sShuttle1Locked)
        OR ("DB_LoaderShuttle1".sShuttlePosExt AND "DB_WorkingModes".sAuto AND NOT "DB_SonplasMain".sSonplasLoader.sOutCollision);                                            // Shuttle EXT - Ext Loader in safe position
   END_REGION

   REGION Axis06 U2 - Feed Stop
       "LBP_Axis06_U2".A_FDSpStop :=
       ("DB_LoaderShuttle2".sShuttlePosExt AND "DB_LoaderAxis".iU2PosSetPoint > "DB_AxisPosMachinePLC".Axis_U2.ExtGateExt AND NOT "DB_DigitalInputs".sExternalGateOpened.sSWStatus)       // Shuttle EXT - Consigne SAS/INT - Sas EXT pas ouvert
       OR ("DB_LoaderShuttle2".sShuttlePosSas AND "DB_LoaderAxis".iU2PosSetPoint < "DB_AxisPosMachinePLC".Axis_U2.IntGateExt AND NOT "DB_DigitalInputs".sExternalGateOpened.sSWStatus)    // Shuttle SAS - Consigne EXT     - Sas EXT pas ouvert
       OR ("DB_LoaderShuttle2".sShuttlePosSas AND "DB_LoaderAxis".iU2PosSetPoint > "DB_AxisPosMachinePLC".Axis_U2.ExtGateInt AND NOT "DB_DigitalInputs".sInternalGateOpened.sSWStatus)    // Shuttle SAS - Consigne INT     - Sas INT pas ouvert
       OR ("DB_LoaderShuttle2".sShuttlePosInt AND "DB_LoaderAxis".iU2PosSetPoint < "DB_AxisPosMachinePLC".Axis_U2.IntGateInt AND NOT "DB_DigitalInputs".sInternalGateOpened.sSWStatus)    // Shuttle INT - Consigne SAS/EXT - Sas INT pas ouvert
       OR ("DB_LoaderShuttle2".sShuttlePosInt AND NOT "DB_LoaderShuttle2".sIntLoaderInSafePos)                                                                                            // Shuttle INT - Int loader in safe position 
       OR ("DB_LoaderShuttle2".sShuttlePosExt AND NOT "DB_LoaderShuttle2".sBwLoaderInSafePos)
       OR ("DB_LoaderShuttle2".sShuttlePosExt AND "DB_BwLoader".sBwCommunication.sShuttle2Locked)
       OR ("DB_LoaderShuttle2".sShuttlePosExt AND "DB_WorkingModes".sAuto AND NOT "DB_SonplasMain".sSonplasLoader.sOutCollision);                                            // Shuttle EXT - Ext Loader in safe position
   END_REGION

   REGION Axis07 V - Feed Stop
       "LBP_Axis07_V".A_FDSpStop := "DB_ExtraMissingPart".sGlobalExtraMissing;
   END_REGION

   REGION Axis08 W - Feed Stop
       "LBP_Axis08_W".A_FDSpStop := "DB_ExtraMissingPart".sGlobalExtraMissing;
   END_REGION

   REGION Check if Key Safety Stop pressed 
       IF "LBP_ModeGroup".E_JOG AND
           "DB_PowerOn".sMachinePower AND
           ("DB_McpKeyboardSignals".sK6_SITestStop.sKeySWStatus
           OR "DB_HmiKeyboardSignals".sK6_SITestStop.sKeySWStatus) THEN
           #sTestStopRequested := true;
           #sTestStopStart := false;
           #sTestStopDone := false;
           #sTestStopError := false;
       END_IF;

   END_REGION

   REGION Dynamisation forced procedure Checking (Test STOP)
       // Asking dynamisation forced
       IF #sTestStopRequested THEN
           IF ("LBP_Axis01_X".SIC.SW2.TestStopReq OR 
               "LBP_Axis02_Y".SIC.SW2.TestStopReq OR
               "LBP_Axis03_ZM".SIC.SW2.TestStopReq OR
               "LBP_Axis04_B".SIC.SW2.TestStopReq OR
               "LBP_Axis05_U1".SIC.SW2.TestStopReq OR
               "LBP_Axis06_U2".SIC.SW2.TestStopReq OR
               "LBP_Axis07_V".SIC.SW2.TestStopReq OR
               "LBP_Axis08_W".SIC.SW2.TestStopReq OR
               "LBP_Axis09_ZL".SIC.SW2.TestStopReq)
           THEN
               "LBP_Axis01_X".SCC.CW1.TeststopStart := TRUE; 
               "LBP_Axis02_Y".SCC.CW1.TeststopStart := TRUE;
               "LBP_Axis03_ZM".SCC.CW1.TeststopStart := TRUE;
               "LBP_Axis04_B".SCC.CW1.TeststopStart := TRUE;
               "LBP_Axis05_U1".SCC.CW1.TeststopStart := TRUE;
               "LBP_Axis06_U2".SCC.CW1.TeststopStart := TRUE;
               "LBP_Axis07_V".SCC.CW1.TeststopStart := TRUE;
               "LBP_Axis08_W".SCC.CW1.TeststopStart := TRUE;
               "LBP_Axis09_ZL".SCC.CW1.TeststopStart := TRUE;
               #sTestStopStart := TRUE;
           ELSE
               #sTestStopDone := TRUE;
               #"BrakeTest ZM".sStartSBT := TRUE;
               #"BrakeTest ZM".sSBTDone := FALSE;
               #"BrakeTest ZL".sStartSBT := TRUE;
               #"BrakeTest ZL".sSBTDone := FALSE;
           END_IF;
           #sTestStopRequested := FALSE;
       END_IF;

       //Timer dynamisation forced : Begin 
       #sTimerTestStopStart.TON (IN := #sTestStopStart,
       PT := t#500ms);

       //Reset dynamisation forcée
       IF #sTimerTestStopStart.Q THEN
           IF "LBP_Axis01_X".SIC.SW2.TestStopAct AND 
               "LBP_Axis02_Y".SIC.SW2.TestStopAct AND
               "LBP_Axis03_ZM".SIC.SW2.TestStopAct AND
               "LBP_Axis04_B".SIC.SW2.TestStopAct AND
               "LBP_Axis05_U1".SIC.SW2.TestStopAct AND
               "LBP_Axis06_U2".SIC.SW2.TestStopAct AND
               "LBP_Axis07_V".SIC.SW2.TestStopAct AND
               "LBP_Axis08_W".SIC.SW2.TestStopAct AND
               "LBP_Axis09_ZL".SIC.SW2.TestStopAct 
           THEN
               "LBP_Axis01_X".SCC.CW1.TeststopStart := FALSE;
               "LBP_Axis02_Y".SCC.CW1.TeststopStart := FALSE;
               "LBP_Axis03_ZM".SCC.CW1.TeststopStart := FALSE;
               "LBP_Axis04_B".SCC.CW1.TeststopStart := FALSE;
               "LBP_Axis05_U1".SCC.CW1.TeststopStart := FALSE;
               "LBP_Axis06_U2".SCC.CW1.TeststopStart := FALSE;
               "LBP_Axis07_V".SCC.CW1.TeststopStart := FALSE;
               "LBP_Axis08_W".SCC.CW1.TeststopStart := FALSE;
               "LBP_Axis09_ZL".SCC.CW1.TeststopStart := FALSE;

               #sTestStopEnd := TRUE;
               #sTestStopStart := FALSE;
           END_IF;
       END_IF;

       //Timer dynamisation forced : End 
       #sTimerTestStopEnd.TON (IN := #sTestStopEnd,
       PT := t#500ms);

       IF #sTimerTestStopEnd.Q THEN

           IF "LBP_Axis01_X".SIC.SW2.TestStopReq         
               OR "LBP_Axis02_Y".SIC.SW2.TestStopReq
               OR "LBP_Axis03_ZM".SIC.SW2.TestStopReq
               OR "LBP_Axis04_B".SIC.SW2.TestStopReq
               OR "LBP_Axis05_U1".SIC.SW2.TestStopReq
               OR "LBP_Axis06_U2".SIC.SW2.TestStopReq
               OR "LBP_Axis07_V".SIC.SW2.TestStopReq
               OR "LBP_Axis08_W".SIC.SW2.TestStopReq
               OR "LBP_Axis09_ZL".SIC.SW2.TestStopReq
           THEN
               #sTestStopError := TRUE;
           END_IF;
           #sTestStopEnd := FALSE;
           #sTestStopDone := TRUE;

           #"BrakeTest ZM".sStartSBT := TRUE;
           #"BrakeTest ZM".sSBTDone := FALSE;
           #"BrakeTest ZL".sStartSBT := TRUE;
           #"BrakeTest ZL".sSBTDone := FALSE;
       END_IF;

       "LBP_AlarmMsgs".UserA[5].A70UUxx[43] := #sTestStopError;  // Msg 700543 : SAFETY: TEST STOP ERROR

       IF "MCP1_In".reset THEN
           "LBP_Axis01_X".SCC.CW1.TeststopStart := FALSE; 
           "LBP_Axis02_Y".SCC.CW1.TeststopStart := FALSE;
           "LBP_Axis03_ZM".SCC.CW1.TeststopStart := FALSE;
           "LBP_Axis04_B".SCC.CW1.TeststopStart := FALSE;
           "LBP_Axis05_U1".SCC.CW1.TeststopStart := FALSE;
           "LBP_Axis06_U2".SCC.CW1.TeststopStart := FALSE;
           "LBP_Axis07_V".SCC.CW1.TeststopStart := FALSE;
           "LBP_Axis08_W".SCC.CW1.TeststopStart := FALSE;
           "LBP_Axis09_ZL".SCC.CW1.TeststopStart := FALSE;

           #sTestStopRequested := FALSE;
           #sTestStopStart := FALSE;
       END_IF;
   END_REGION

   REGION Safe Brake Test Control (SBT) - Z axis

       IF "MCP1_In".reset OR NOT "LBP_ModeGroup".E_JOG THEN
           #"BrakeTest ZM".sStartSBT := FALSE;
           #"BrakeTest ZL".sStartSBT := FALSE;
       END_IF;

       #"sBrakeTest ZM"(iStartBt := #"BrakeTest ZM".sStartSBT,
                   iQuit := "MCP1_In".reset,
                   iExternalBrakeClosed := false,
                   iMaxStepTime := T#10S,
                   iBrakeNum := false,
                   iActivateAutoDirection := false,
                   iSetManualDirection := false,
                   iTestSequence := false,
                   oCloseExternalBrake => #"BrakeTest ZM".scloseExternalBrake,
                   oDone => #"BrakeTest ZM".sDone,
                   oError => #"BrakeTest ZM".sError,
                   oStateNum => #"BrakeTest ZM".sStateNum,
                   oDiagnoseError => #"BrakeTest ZM".sDiagnoseError,
                   oError1 => #sErrorN[1],
                   oError2 => #sErrorN[2],
                   oError3 => #sErrorN[3],
                   oError4 => #sErrorN[4],
                   oError5 => #sErrorN[5],
                   oError6 => #sErrorN[6],
                   oError7 => #sErrorN[7],
                   oError8 => #sErrorN[8],
                   ioAxisDB := "LBP_Axis03_ZM");

   #"sBrakeTest ZL"(iStartBt := #"BrakeTest ZL".sStartSBT,
                     iQuit := "MCP1_In".reset,
                     iExternalBrakeClosed := false,
                     iMaxStepTime := T#10S,
                     iBrakeNum := false,
                     iActivateAutoDirection := false,
                     iSetManualDirection := false,
                     iTestSequence := false,
                     oCloseExternalBrake => #"BrakeTest ZL".scloseExternalBrake,
                     oDone => #"BrakeTest ZL".sDone,
                     oError => #"BrakeTest ZL".sError,
                     oStateNum => #"BrakeTest ZL".sStateNum,
                     oDiagnoseError => #"BrakeTest ZL".sDiagnoseError,
                     oError1 => #sErrorN[1],
                     oError2 => #sErrorN[2],
                     oError3 => #sErrorN[3],
                     oError4 => #sErrorN[4],
                     oError5 => #sErrorN[5],
                     oError6 => #sErrorN[6],
                     oError7 => #sErrorN[7],
                     oError8 => #sErrorN[8],
                     ioAxisDB := "LBP_Axis09_ZL");

    IF #"BrakeTest ZM".sDone AND #"BrakeTest ZL".sDone THEN
        #"BrakeTest ZM".sStartSBT := FALSE;
        #"BrakeTest ZM".sSBTDone := TRUE;
        #"BrakeTest ZL".sStartSBT := FALSE;
        #"BrakeTest ZL".sSBTDone := TRUE;
           "LBP_AlarmMsgs".UserA[5].A70UUxx[12] := FALSE;  // Msg 700512 "SAFETY: THE BRAKE TEST IS NOT WORKING, PLEASE RESET"
       END_IF;

       IF #"BrakeTest ZM".sDiagnoseError <> 0 AND #"BrakeTest ZL".sDiagnoseError <> 0 THEN
           "LBP_AlarmMsgs".UserA[5].A70UUxx[12] := TRUE;  // Msg 700512 "SAFETY: THE BRAKE TEST IS NOT WORKING, PLEASE RESET"
       END_IF;

   END_REGION

   REGION LED SAFETY TEST 
       #sLedSITestSlowFlashing :=
       "LBP_ModeGroup".E_JOG
       AND "DB_PowerOn".sMachinePower
       AND NOT #"BrakeTest ZM".sStartSBT
       AND NOT #"BrakeTest ZL".sStartSBT
       AND NOT #sTestStopStart
       AND "DB_DataFromSafety".DoorsClosed
       AND (NOT #"BrakeTest ZM".sSBTDone
           OR NOT #"BrakeTest ZL".sSBTDone
           OR NOT #sTestStopDone
           OR "LBP_Axis01_X".SIC.SW2.TestStopReq     
           OR "LBP_Axis02_Y".SIC.SW2.TestStopReq
           OR "LBP_Axis03_ZM".SIC.SW2.TestStopReq
           OR "LBP_Axis04_B".SIC.SW2.TestStopReq
           OR "LBP_Axis05_U1".SIC.SW2.TestStopReq
           OR "LBP_Axis06_U2".SIC.SW2.TestStopReq
           OR "LBP_Axis07_V".SIC.SW2.TestStopReq
           OR "LBP_Axis08_W".SIC.SW2.TestStopReq
           OR "LBP_Axis09_ZL".SIC.SW2.TestStopReq);
       #sLedSITestQuickFlashing :=
       ("LBP_AlarmMsgs".UserA[5].A70UUxx[12]              // Msg 700512 "SAFETY: THE BRAKE TEST IS NOT WORKING, PLEASE RESET"
           OR "LBP_AlarmMsgs".UserA[5].A70UUxx[43])       // Msg 700543 "SAFETY: TEST STOP ERROR"
           AND "DB_PowerOn".sMachinePower;

       #sLedSITestOK :=
       NOT #"BrakeTest ZM".sStartSBT
           AND NOT  #"BrakeTest ZL".sStartSBT
           AND NOT #sTestStopStart
           AND NOT "LBP_AlarmMsgs".UserA[5].A70UUxx[12]   // Msg 700512 "SAFETY: THE BRAKE TEST IS NOT WORKING, PLEASE RESET"
           AND NOT "LBP_AlarmMsgs".UserA[5].A70UUxx[43]   // Msg 700543 "SAFETY: TEST STOP ERROR"
           AND #"BrakeTest ZM".sSBTDone
           AND #"BrakeTest ZL".sSBTDone
           AND #sTestStopDone
           AND NOT #sLedSITestSlowFlashing
           AND NOT #sLedSITestQuickFlashing;

           "DB_McpKeyboardSignals".sK6_SITestStop.sLedSWStatus :=     
           #sLedSITestOK
           OR (#sLedSITestSlowFlashing AND "Clock_1Hz")
           OR (#sLedSITestQuickFlashing AND "Clock_2Hz");

           "DB_HmiKeyboardSignals".sK6_SITestStop.sLedSWStatus :=
           #sLedSITestOK
           OR (#sLedSITestSlowFlashing AND "Clock_1Hz")
           OR (#sLedSITestQuickFlashing AND "Clock_2Hz");
   END_REGION
END_FUNCTION_BLOCK

FUNCTION_BLOCK "FB_BrakeTest"   // FB412, SCL
TITLE = BrakeTest
{ S7_Optimized_Access := 'FALSE' }
VERSION : 3.12
// Sinamics brake test
// stored: AutoNumber false, IsIECCheckEnabled true, SetENOAutomatically false
   VAR_INPUT
      iStartBt : Bool;   // start BT (Bit must only be resetted as soon as done = 1)
      iQuit : Bool;   // quit error
      iExternalBrakeClosed : Bool;   // feedback external brake; if closed = 1, if open = 0
      iMaxStepTime : Time := T#6S;   // max time per sequencer step
      iBrakeNum : Bool;   // number of brake to be tested; brake 1 = 0; brake 2 = 1
      iActivateAutoDirection : Bool;   // enable automatic detection of direction of test torque
      iSetManualDirection : Bool;   // manual selection of direction of test torque
      iTestSequence : Bool;   // selection of test sequence; sequence 1 = 0, sequence 2 = 1
   END_VAR
   VAR_OUTPUT
      oCloseExternalBrake : Bool;   // signal to close the external brake; close = 1, open = 0
      oDone : Bool;   // done without errors
      oError : Bool;   // error occurred
      oStateNum : Int;   // active step of the sequence
      oDiagnoseError : Int;   // error number
      oError1 : Bool;   // invalid sequence step
      oError2 : Bool;   // invalid start condition: axis not stationery
      oError3 : Bool;   // invalid start condition: pulse enable missing
      oError4 : Bool;   // brake test noch successful
      oError5 : Bool;   // sequence step time monitoring error
      oError6 : Bool;   // startBT reset while in progress
      oError7 : Bool;   // invalid error number
      oError8 : Bool;   // no feedback external brake within "maxStepTime"
   END_VAR
   VAR_IN_OUT
      ioAxisDB : "LBP_typeAxisX";   // UDT of test axis (has to be connected!)
   END_VAR
   VAR
      sStepNum : Int;   // active sequencer step
      sEdgeFlagStop : Bool;   // falling edge flag of startBT
      sEdgeFlagStart : Bool;   // rising edge flag of startBT
      sStepNumOld : Int;   // sequencer step of the previous PLC cycle
      sBTDeselectionDelay : Bool;   // TOF, Q output of deselection timer
      sStartTimer { ExternalVisible := 'False'; ExternalWritable := 'False'} : Bool := true;   // start timer of sequencer time monitoring
      sActiveError : Bool;   // active error
      sInstIecTimerTimeStepBt { S7_SetPoint := 'True'} : TOF_TIME;   // timer for monitoring the steps of the sequencer
      sInstIecTimerSelectSafeBt { S7_SetPoint := 'True'} : TOF_TIME;   // timer to delay the program, if BT is deselected
      sErrorNum { ExternalVisible := 'False'; ExternalWritable := 'False'} : Int;   // provisional error number
   END_VAR
   VAR_TEMP
      tIncrement : Bool;   // increment sequencer
      tTimeSig : Bool;   // TOF, Q output sequencer time monitoring
      tRisBTStart : Bool;   // rising edge startBT
      tFalBTStart : Bool;   // falling edge startBT
      tErr6 : Bool;   // error no. 6
   END_VAR
BEGIN
   REGION BLOCK INFO HEADER
   //=============================================================================
   // Siemens
   // (c)Copyright 2021 All Rights Reserved
   // ----------------------------------------------------------------------------
   // Library:       Lib_SBT_SINUMERIK_ONE
   // Tested with:   V6.13 / NCU 1760
   // Engineering:   TIA Portal V16 Update 4
   // Restrictions:  -
   // Requirements:  motor with brake; UDT "LBP_typeAxisX" of the axis to be tested
   // Functionality: brake test for safety axis
   // ----------------------------------------------------------------------------
   // Change log table:
   // Version   Date         Expert in charge   Changes applied
   // 03.01.02  01.12.2021   Siemens AG         First released version
   // =============================================================================
   END_REGION BLOCK INFO HEADER

   REGION set temp variables 
     #tErr6 := 0;
     #tIncrement := 0;
     #tTimeSig := 0;
     #tRisBTStart := 0;
     #tFalBTStart := 0;
   END_REGION

   REGION edge evaluation 
     // rising edge startBt 
     #tRisBTStart := (#iStartBt AND NOT #iQuit) AND NOT #sEdgeFlagStart;
     #sEdgeFlagStart := (#iStartBt AND NOT #iQuit);

     // falling edge startBt 
     #tFalBTStart := NOT #iStartBt AND #sEdgeFlagStop;
     #sEdgeFlagStop := #iStartBt;
   END_REGION

   REGION return function if Test is inactive 
     // return function while Test is inactive 
     IF NOT (#iStartBt OR #tFalBTStart OR #tRisBTStart OR
       #sActiveError OR #iQuit) THEN
       RETURN;
   END_IF;
   END_REGION

   REGION reset brake test enable when FB stopped 
     IF NOT (#iStartBt OR #sActiveError) THEN
       IF #sStepNum <> 0 THEN
         //error number 6: SBT is cancelled with startBt=0 
         #tErr6 := 1;
       END_IF;
       //stop step sequence 
       #sStepNum := 0;
       //Cancellation/deselection SBT 
       #ioAxisDB.A_StartBrakeTest := 0;
       #ioAxisDB.SCC.CW3.SelectionSBT := 0;
       #ioAxisDB.SCC.CW3.BT_Start := 0;
     END_IF;
   END_REGION

   REGION external brake status/control 
     IF #iStartBt THEN
       //control external brake 
       #oCloseExternalBrake := #ioAxisDB.SIC.SW3.BrakeReq;
       //status external brake 
       #ioAxisDB.SCC.CW3.BrakeClosed := #iExternalBrakeClosed;
     END_IF;

   END_REGION

   REGION timer 
     //start Watchdog Timer on the beginning and for every new step 
     #sStartTimer := 0;
     IF (#sStepNum <> #sStepNumOld)
       OR (#tRisBTStart = 1) THEN
       #sStartTimer := 1;
     END_IF;

     // Timer (TOF) Time delay stop SBT 
     #sInstIecTimerSelectSafeBt(IN := #ioAxisDB.A_StartBrakeTest,
                               PT := T#100ms,
                               Q => #sBTDeselectionDelay);

     // Timer (TOF) Watchdog for step sequence  
     #sInstIecTimerTimeStepBt(IN := #sStartTimer,
                             PT := #iMaxStepTime,
                             Q => #tTimeSig);
     #sStepNumOld := #sStepNum;
   END_REGION

   REGION step sequence 
     //start step sequence with rising Edge startBt 
     IF #tRisBTStart THEN
       #sStepNum := 1;
     END_IF;

     // step sequence Brake test 
     CASE #sStepNum OF
       0:  // step sequence not running 
         #sActiveError := 0;
         #oError := 0;
         #oDone := 0;
         #sErrorNum := 0;
       1:  // Check start condition 
         IF NOT #ioAxisDB.E_Stat THEN
           //Axis/spindle is not stationary(n < nmin) 
           //Error Number 2 
           #sErrorNum := 2;
         END_IF;
         IF NOT #ioAxisDB.E_PulseEnable OR NOT #ioAxisDB.E_DriveRunEn THEN
           //Pulse or controller enable is missing 
           //Error Number 3 
           #sErrorNum := 3;
         END_IF;
         IF (#sErrorNum = 0) AND #tTimeSig THEN
           #tIncrement := 1; //next Step                     
         END_IF;

       2:  //Select Brake 1 OR 2 
         #ioAxisDB.SCC.CW3.Brake_1_2 := #iBrakeNum;
         IF #tTimeSig = 1 THEN
           #tIncrement := 1;//next Step  
         END_IF;

       3:  //Select Test sequence 1 or 2 
         #ioAxisDB.SCC.CW3.Testseq_1_2 := #iTestSequence;
         IF #tTimeSig = 1 THEN
           #tIncrement := 1;//next Step  
         END_IF;

       4:  //Set NCK Start signal for Brake test 
         #ioAxisDB.A_StartBrakeTest := 1;
         //feedback NCK Brake test active #axisDB.E_BrakeTest 
         IF (#ioAxisDB.E_BrakeTest) AND (#tTimeSig) THEN
           #tIncrement := 1;//next Step  
         END_IF;

       5:  // Select SBT  
         #ioAxisDB.SCC.CW3.SelectionSBT := 1;
         //feedback SBT selected #axisDB.SIC.SW3.SBT_Sel and test torque from drive #axisDB.SIC.SW3.SetpSettingDrive 
         IF (#tTimeSig = 1) AND #ioAxisDB.SIC.SW3.SBT_Sel AND #ioAxisDB.SIC.SW3.SetpSettingDrive THEN
           #tIncrement := 1;//next Step  
         END_IF;
       6: //Select manual or auto direction  
         IF #iActivateAutoDirection = 1 THEN
           //auto direction 
           #ioAxisDB.SCC.CW3.DirOfROT := #ioAxisDB.SIC.SW3.SignLoadTorque;
         ELSE
           //Manual direction  
           // #setManualDirection=false negative direction 
           // #setManualDirection=true positive direction 
           #ioAxisDB.SCC.CW3.DirOfROT := #iSetManualDirection;
         END_IF;

         IF #tTimeSig = 1 THEN
           #tIncrement := 1;//next Step  
         END_IF;

       7:  // Request start Brake test SCC 
         #ioAxisDB.SCC.CW3.BT_Start := 1;
         //feedback Brake test active SIC #axisDB.SIC.SW3.BT_Act 
         IF #ioAxisDB.SIC.SW3.BT_Act AND #tTimeSig THEN
           #tIncrement := 1;//next Step  
         END_IF;
       8: //Check if the condition of the external brake fits the request 
         IF ((#ioAxisDB.SIC.SW3.BrakeReq XOR #ioAxisDB.SCC.CW3.BrakeClosed) AND (NOT #tTimeSig)) THEN
           //Error external Brake 
           #sErrorNum := 8;
         END_IF;

         IF (#ioAxisDB.SIC.SW3.BrakeReq = #ioAxisDB.SCC.CW3.BrakeClosed) AND #tTimeSig THEN

           #tIncrement := 1;//next Step  
         END_IF;

       9:  // Waiting for SBT finished signal 
         IF #ioAxisDB.SIC.SW3.BT_Finished AND #tTimeSig THEN
           #tIncrement := 1;//next Step  
         END_IF;
       10: // Check if SBT was OK 
         IF NOT (#ioAxisDB.SIC.SW3.BT_Finished AND #ioAxisDB.SIC.SW3.BT_OK) THEN
           //SBT finished with error 
           #sErrorNum := 4;
         END_IF;
         IF #tTimeSig AND #ioAxisDB.SIC.SW3.BT_OK THEN
           #tIncrement := 1;//next Step  
         END_IF;
       11: // Request stop Brake test SCC 
         #ioAxisDB.SCC.CW3.BT_Start := 0;
         IF #tTimeSig AND NOT (#ioAxisDB.SIC.SW3.BT_Act AND #sBTDeselectionDelay) THEN
           //Feedback SIC SBT is stopped  
           #tIncrement := 1;//next Step  
         END_IF;
       12: // Reset NCK Start signal for Brake test 
         // Deselect SBT via SCC 
         #ioAxisDB.A_StartBrakeTest := 0;
         #ioAxisDB.SCC.CW3.SelectionSBT := 0;
         IF #tTimeSig AND NOT #ioAxisDB.E_BrakeTest AND NOT #ioAxisDB.SIC.SW3.SBT_Sel THEN
           // SBT finished without error 
           // set done 
           // stop step sequence 
           #sStepNum := 0;
           #oDone := 1;
         END_IF;
       ELSE:
         //wrong step number 
         #sErrorNum := 1;
   END_CASE;
   END_REGION

   REGION error handling 
     // error number 6: SBT is cancelled with startBt=0 while running without error 
     IF #tErr6 THEN
       //Error Number 6 
       #sErrorNum := 6;
       //set error 
       #oError := 1;
     END_IF;

     // Watchdog step sequence -> Error Num 5 
     IF #sErrorNum = 0 AND (#sStepNum <> 0) AND NOT #tTimeSig THEN
       #sErrorNum := 5;
       #oError := 1;
       #sActiveError := 1;
     END_IF;

     // Error Bit 
     CASE #sErrorNum OF
       0:
         ;
       1:
         #oError1 := 1;
       2:
         #oError2 := 1;
       3:
         #oError3 := 1;
       4:
         #oError4 := 1;
       5:
         #oError5 := 1;
       6:
         #oError6 := 1;
       8:
         #oError8 := 1;
       ELSE                  // Wrong error number -> set Error Num 7
         #oError7 := 1;
         #sErrorNum := 7;
     END_CASE;

     // output error number and step number for diagnose 
     IF #sErrorNum <> 0 THEN
         #oError := 1;
         #sActiveError := 1;
         #oDiagnoseError := #sErrorNum;
         #oStateNum := #sStepNum;
     END_IF;
   END_REGION

   REGION quit error 
     //reset signals  
       IF #iQuit = 1 THEN
           #ioAxisDB.SCC.CW3.BT_Start := 0;
           #ioAxisDB.A_StartBrakeTest := 0;
           #ioAxisDB.SCC.CW3.Brake_1_2 := 0;
           #ioAxisDB.SCC.CW3.SelectionSBT := 0;
           #oCloseExternalBrake := 0;
           #sStartTimer := 1;
           #oError := 0;
           #oError1 := 0;
           #oError2 := 0;
           #oError3 := 0;
           #oError4 := 0;
           #oError5 := 0;
           #oError6 := 0;
           #oError7 := 0;
           #oError8 := 0;
           #sActiveError := 0;
           #oDiagnoseError := 0;
           #oStateNum := 0;
           #sStepNum := 0;
           #tIncrement := 0;
       END_IF;
   END_REGION

   REGION increment step sequence 
     //increment step number 
     IF #sErrorNum = 0 AND #tIncrement = 1 THEN
       //increment step number 
       #sStepNum += 1;
       //update output step number 
       #oStateNum := #sStepNum;
   END_IF;
   END_REGION
END_FUNCTION_BLOCK

FUNCTION_BLOCK "FB_AxisPosition"   // FB411, SCL
{ S7_Optimized_Access := 'TRUE' }
// stored: AutoNumber false, MemoryReserve 100, SetENOAutomatically false
   VAR
      sError { ExternalAccessible := 'False'; ExternalVisible := 'False'; ExternalWritable := 'False'} : Bool;
      sNDR { ExternalAccessible := 'False'; ExternalVisible := 'False'; ExternalWritable := 'False'} : Bool;
      sState { ExternalAccessible := 'False'; ExternalVisible := 'False'; ExternalWritable := 'False'} : Word;
      sAxis01_X : Struct
         "$AA_IM" : LReal;
         "$MA_POS_LIMIT_MINUS" : LReal;
         "$MA_POS_LIMIT_MINUS2" : LReal;
         "$MA_POS_LIMIT_PLUS" : LReal;
         "$MA_POS_LIMIT_PLUS2" : LReal;
         "$MA_JOG_VELO" : LReal;
         "$MA_JOG_VELO_RAPID" : LReal;
         "$MA_MAX_AX_VELO" : LReal;
         "$A1_M_FP_POS4_30600" : LReal;
      END_STRUCT;
      sAxis02_Y : Struct
         "$AA_IM" : LReal;
         "$MA_POS_LIMIT_MINUS" : LReal;
         "$MA_POS_LIMIT_MINUS2" : LReal;
         "$MA_POS_LIMIT_PLUS" : LReal;
         "$MA_POS_LIMIT_PLUS2" : LReal;
         "$MA_JOG_VELO" : LReal;
         "$MA_JOG_VELO_RAPID" : LReal;
         "$MA_MAX_AX_VELO" : LReal;
      END_STRUCT;
      sAxis03_ZM : Struct
         "$AA_IM" : LReal;
         "$MA_POS_LIMIT_MINUS" : LReal;
         "$MA_POS_LIMIT_MINUS2" : LReal;
         "$MA_POS_LIMIT_PLUS" : LReal;
         "$MA_POS_LIMIT_PLUS2" : LReal;
         "$MA_JOG_VELO" : LReal;
         "$MA_JOG_VELO_RAPID" : LReal;
         "$MA_MAX_AX_VELO" : LReal;
      END_STRUCT;
      sAxis04_B : Struct
         "$AA_IM" : LReal;
         "$MA_POS_LIMIT_MINUS" : LReal;
         "$MA_POS_LIMIT_MINUS2" : LReal;
         "$MA_POS_LIMIT_PLUS" : LReal;
         "$MA_POS_LIMIT_PLUS2" : LReal;
         "$MA_JOG_VELO" : LReal;
         "$MA_JOG_VELO_RAPID" : LReal;
         "$MA_MAX_AX_VELO" : LReal;
      END_STRUCT;
      sAxis05_U1 : Struct
         "$AA_IM" : LReal;
         "$MA_POS_LIMIT_MINUS" : LReal;
         "$MA_POS_LIMIT_MINUS2" : LReal;
         "$MA_POS_LIMIT_PLUS" : LReal;
         "$MA_POS_LIMIT_PLUS2" : LReal;
         "$MA_JOG_VELO" : LReal;
         "$MA_JOG_VELO_RAPID" : LReal;
         "$MA_MAX_AX_VELO" : LReal;
      END_STRUCT;
      sAxis06_U2 : Struct
         "$AA_IM" : LReal;
         "$MA_POS_LIMIT_MINUS" : LReal;
         "$MA_POS_LIMIT_MINUS2" : LReal;
         "$MA_POS_LIMIT_PLUS" : LReal;
         "$MA_POS_LIMIT_PLUS2" : LReal;
         "$MA_JOG_VELO" : LReal;
         "$MA_JOG_VELO_RAPID" : LReal;
         "$MA_MAX_AX_VELO" : LReal;
         "$A1_M_FP_POS2_30600" : LReal;
      END_STRUCT;
      sAxis07_V : Struct
         "$AA_IM" : LReal;
         "$MA_POS_LIMIT_MINUS" : LReal;
         "$MA_POS_LIMIT_MINUS2" : LReal;
         "$MA_POS_LIMIT_PLUS" : LReal;
         "$MA_POS_LIMIT_PLUS2" : LReal;
         "$MA_JOG_VELO" : LReal;
         "$MA_JOG_VELO_RAPID" : LReal;
         "$MA_MAX_AX_VELO" : LReal;
      END_STRUCT;
      sAxis08_W : Struct
         "$AA_IM" : LReal;
         "$MA_POS_LIMIT_MINUS" : LReal;
         "$MA_POS_LIMIT_MINUS2" : LReal;
         "$MA_POS_LIMIT_PLUS" : LReal;
         "$MA_POS_LIMIT_PLUS2" : LReal;
         "$MA_JOG_VELO" : LReal;
         "$MA_JOG_VELO_RAPID" : LReal;
         "$MA_MAX_AX_VELO" : LReal;
      END_STRUCT;
      sAxis09_ZL : Struct
         "$AA_IM" : LReal;
         "$MA_POS_LIMIT_MINUS" : LReal;
         "$MA_POS_LIMIT_MINUS2" : LReal;
         "$MA_POS_LIMIT_PLUS" : LReal;
         "$MA_POS_LIMIT_PLUS2" : LReal;
         "$MA_JOG_VELO" : LReal;
         "$MA_JOG_VELO_RAPID" : LReal;
         "$MA_MAX_AX_VELO" : LReal;
      END_STRUCT;
   END_VAR
BEGIN
   REGION Description header 
       //==================================================================================
       // POSALUX Swiss SA / (C) Copyright 2025
       //----------------------------------------------------------------------------------
       // Title: FB_AxisPosition
       // Comment/Function: These function blocks allow reading NC data related to 
       //                   axis positions, references, and speeds from the NC.
       // Author: Fabien WALDT
       // Engineering: TIA Portal v17
       //----------------------------------------------------------------------------------
       // Change log table:
       // Version  | Date     | Expert in charge | Changes applied
       // ---------|----------|------------------|------------------------------------
       // 00.00.01 | 20250423 | WFA              | First released version
       // ==================================================================================
   END_REGION

   REGION Axis 01 X
       "LBP_ReadVar_DB_Axis01_X"(Req := "Clock_10Hz",
                                 NumVar := 8,
                                 Addr1 := "DB_NcVarSelect_AA_IM"."$AA_IM_Axis01_X".token,
                                 Addr2 := "DB_NcVarSelect_MA_POS_LIMIT_MINUS"."$MA_POS_LIMIT_MINUS_Axis01_X".token,
                                 Addr3 := "DB_NcVarSelect_MA_POS_LIMIT_MINUS2"."$MA_POS_LIMIT_MINUS2_Axis01_X".token,
                                 Addr4 := "DB_NcVarSelect_MA_POS_LIMIT_PLUS"."$MA_POS_LIMIT_PLUS_Axis01_X".token,
                                 Addr5 := "DB_NcVarSelect_MA_POS_LIMIT_PLUS2"."$MA_POS_LIMIT_PLUS2_Axis01_X".token,
                                 Addr6 := "DB_NcVarSelect_MA_JOG_VELO"."$MA_JOG_VELO_Axis01_X".token,
                                 Addr7 := "DB_NcVarSelect_MA_JOG_VELO_RAPID"."$MA_JOG_VELO_RAPID_Axis01_X".token,
                                 Addr8 := "DB_NcVarSelect_M_MAX_AX_VELO"."$MA_JOG_VELO_Axis01_X".token,
                                 Error => #sError,
                                 NDR => #sNDR,
                                 State => #sState,
                                 RD1 := #sAxis01_X."$AA_IM",
                                 RD2 := #sAxis01_X."$MA_POS_LIMIT_MINUS",
                                 RD3 := #sAxis01_X."$MA_POS_LIMIT_MINUS2",
                                 RD4 := #sAxis01_X."$MA_POS_LIMIT_PLUS",
                                 RD5 := #sAxis01_X."$MA_POS_LIMIT_PLUS2",
                                 RD6 := #sAxis01_X."$MA_JOG_VELO",
                                 RD7 := #sAxis01_X."$MA_JOG_VELO_RAPID",
                                 RD8 := #sAxis01_X."$MA_MAX_AX_VELO");
   END_REGION

   REGION Axis 02 Y
       "LBP_ReadVar_DB_Axis02_Y"(Req := "Clock_10Hz",
                                 NumVar := 8,
                                 Addr1 := "DB_NcVarSelect_AA_IM"."$AA_IM_Axis02_Y".token,
                                 Addr2 := "DB_NcVarSelect_MA_POS_LIMIT_MINUS"."$MA_POS_LIMIT_MINUS_Axis02_Y".token,
                                 Addr3 := "DB_NcVarSelect_MA_POS_LIMIT_MINUS2"."$MA_POS_LIMIT_MINUS2_Axis02_Y".token,
                                 Addr4 := "DB_NcVarSelect_MA_POS_LIMIT_PLUS"."$MA_POS_LIMIT_PLUS_Axis02_Y".token,
                                 Addr5 := "DB_NcVarSelect_MA_POS_LIMIT_PLUS2"."$MA_POS_LIMIT_PLUS2_Axis02_Y".token,
                                 Addr6 := "DB_NcVarSelect_MA_JOG_VELO"."$MA_JOG_VELO_Axis02_Y".token,
                                 Addr7 := "DB_NcVarSelect_MA_JOG_VELO_RAPID"."$MA_JOG_VELO_RAPID_Axis02_Y".token,
                                 Addr8 := "DB_NcVarSelect_M_MAX_AX_VELO"."$MA_JOG_VELO_Axis02_Y".token,
                                 Error => #sError,
                                 NDR => #sNDR,
                                 State => #sState,
                                 RD1 := #sAxis02_Y."$AA_IM",
                                 RD2 := #sAxis02_Y."$MA_POS_LIMIT_MINUS",
                                 RD3 := #sAxis02_Y."$MA_POS_LIMIT_MINUS2",
                                 RD4 := #sAxis02_Y."$MA_POS_LIMIT_PLUS",
                                 RD5 := #sAxis02_Y."$MA_POS_LIMIT_PLUS2",
                                 RD6 := #sAxis02_Y."$MA_JOG_VELO",
                                 RD7 := #sAxis02_Y."$MA_JOG_VELO_RAPID",
                                 RD8 := #sAxis02_Y."$MA_MAX_AX_VELO");
   END_REGION

   REGION Axis 03 ZM
       "LBP_ReadVar_DB_Axis03_ZM"(Req := "Clock_10Hz",
                                  NumVar := 8,
                                  Addr1 := "DB_NcVarSelect_AA_IM"."$AA_IM_Axis03_ZM".token,
                                  Addr2 := "DB_NcVarSelect_MA_POS_LIMIT_MINUS"."$MA_POS_LIMIT_MINUS_Axis03_ZM".token,
                                  Addr3 := "DB_NcVarSelect_MA_POS_LIMIT_MINUS2"."$MA_POS_LIMIT_MINUS2_Axis03_ZM".token,
                                  Addr4 := "DB_NcVarSelect_MA_POS_LIMIT_PLUS"."$MA_POS_LIMIT_PLUS_Axis03_ZM".token,
                                  Addr5 := "DB_NcVarSelect_MA_POS_LIMIT_PLUS2"."$MA_POS_LIMIT_PLUS2_Axis03_ZM".token,
                                  Addr6 := "DB_NcVarSelect_MA_JOG_VELO"."$MA_JOG_VELO_Axis03_ZM".token,
                                  Addr7 := "DB_NcVarSelect_MA_JOG_VELO_RAPID"."$MA_JOG_VELO_RAPID_Axis03_ZM".token,
                                  Addr8 := "DB_NcVarSelect_M_MAX_AX_VELO"."$MA_JOG_VELO_Axis03_ZM".token,
                                  Error => #sError,
                                  NDR => #sNDR,
                                  State => #sState,
                                  RD1 := #sAxis03_ZM."$AA_IM",
                                  RD2 := #sAxis03_ZM."$MA_POS_LIMIT_MINUS",
                                  RD3 := #sAxis03_ZM."$MA_POS_LIMIT_MINUS2",
                                  RD4 := #sAxis03_ZM."$MA_POS_LIMIT_PLUS",
                                  RD5 := #sAxis03_ZM."$MA_POS_LIMIT_PLUS2",
                                  RD6 := #sAxis03_ZM."$MA_JOG_VELO",
                                  RD7 := #sAxis03_ZM."$MA_JOG_VELO_RAPID",
                                  RD8 := #sAxis03_ZM."$MA_MAX_AX_VELO");
   END_REGION

   REGION Axis 04 B
       "LBP_ReadVar_DB_Axis04_B"(Req := "Clock_10Hz",
                                 NumVar := 8,
                                 Addr1 := "DB_NcVarSelect_AA_IM"."$AA_IM_Axis04_B".token,
                                 Addr2 := "DB_NcVarSelect_MA_POS_LIMIT_MINUS"."$MA_POS_LIMIT_MINUS_Axis04_B".token,
                                 Addr3 := "DB_NcVarSelect_MA_POS_LIMIT_MINUS2"."$MA_POS_LIMIT_MINUS2_Axis04_B".token,
                                 Addr4 := "DB_NcVarSelect_MA_POS_LIMIT_PLUS"."$MA_POS_LIMIT_PLUS_Axis04_B".token,
                                 Addr5 := "DB_NcVarSelect_MA_POS_LIMIT_PLUS2"."$MA_POS_LIMIT_PLUS2_Axis04_B".token,
                                 Addr6 := "DB_NcVarSelect_MA_JOG_VELO"."$MA_JOG_VELO_Axis04_B".token,
                                 Addr7 := "DB_NcVarSelect_MA_JOG_VELO_RAPID"."$MA_JOG_VELO_RAPID_Axis04_B".token,
                                 Addr8 := "DB_NcVarSelect_M_MAX_AX_VELO"."$MA_JOG_VELO_Axis04_B".token,
                                 Error => #sError,
                                 NDR => #sNDR,
                                 State => #sState,
                                 RD1 := #sAxis04_B."$AA_IM",
                                 RD2 := #sAxis04_B."$MA_POS_LIMIT_MINUS",
                                 RD3 := #sAxis04_B."$MA_POS_LIMIT_MINUS2",
                                 RD4 := #sAxis04_B."$MA_POS_LIMIT_PLUS",
                                 RD5 := #sAxis04_B."$MA_POS_LIMIT_PLUS2",
                                 RD6 := #sAxis04_B."$MA_JOG_VELO",
                                 RD7 := #sAxis04_B."$MA_JOG_VELO_RAPID",
                                 RD8 := #sAxis04_B."$MA_MAX_AX_VELO");
   END_REGION

   REGION Axis 05 U1
       "LBP_ReadVar_DB_Axis05_U1"(Req := NOT "Clock_10Hz",
                                  NumVar := 8,
                                  Addr1 := "DB_NcVarSelect_AA_IM"."$AA_IM_Axis05_U1".token,
                                  Addr2 := "DB_NcVarSelect_MA_POS_LIMIT_MINUS"."$MA_POS_LIMIT_MINUS_Axis05_U1".token,
                                  Addr3 := "DB_NcVarSelect_MA_POS_LIMIT_MINUS2"."$MA_POS_LIMIT_MINUS2_Axis05_U1".token,
                                  Addr4 := "DB_NcVarSelect_MA_POS_LIMIT_PLUS"."$MA_POS_LIMIT_PLUS_Axis05_U1".token,
                                  Addr5 := "DB_NcVarSelect_MA_POS_LIMIT_PLUS2"."$MA_POS_LIMIT_PLUS2_Axis05_U1".token,
                                  Addr6 := "DB_NcVarSelect_MA_JOG_VELO"."$MA_JOG_VELO_Axis05_U1".token,
                                  Addr7 := "DB_NcVarSelect_MA_JOG_VELO_RAPID"."$MA_JOG_VELO_RAPID_Axis05_U1".token,
                                  Addr8 := "DB_NcVarSelect_M_MAX_AX_VELO"."$MA_JOG_VELO_Axis05_U1".token,
                                  Error => #sError,
                                  NDR => #sNDR,
                                  State => #sState,
                                  RD1 := #sAxis05_U1."$AA_IM",
                                  RD2 := #sAxis05_U1."$MA_POS_LIMIT_MINUS",
                                  RD3 := #sAxis05_U1."$MA_POS_LIMIT_MINUS2",
                                  RD4 := #sAxis05_U1."$MA_POS_LIMIT_PLUS",
                                  RD5 := #sAxis05_U1."$MA_POS_LIMIT_PLUS2",
                                  RD6 := #sAxis05_U1."$MA_JOG_VELO",
                                  RD7 := #sAxis05_U1."$MA_JOG_VELO_RAPID",
                                  RD8 := #sAxis05_U1."$MA_MAX_AX_VELO");
   END_REGION

   REGION Axis 06 U2
       "LBP_ReadVar_DB_Axis06_U2"(Req := NOT "Clock_10Hz",
                                  NumVar := 8,
                                  Addr1 := "DB_NcVarSelect_AA_IM"."$AA_IM_Axis06_U2".token,
                                  Addr2 := "DB_NcVarSelect_MA_POS_LIMIT_MINUS"."$MA_POS_LIMIT_MINUS_Axis06_U2".token,
                                  Addr3 := "DB_NcVarSelect_MA_POS_LIMIT_MINUS2"."$MA_POS_LIMIT_MINUS2_Axis06_U2".token,
                                  Addr4 := "DB_NcVarSelect_MA_POS_LIMIT_PLUS"."$MA_POS_LIMIT_PLUS_Axis06_U2".token,
                                  Addr5 := "DB_NcVarSelect_MA_POS_LIMIT_PLUS2"."$MA_POS_LIMIT_PLUS2_Axis06_U2".token,
                                  Addr6 := "DB_NcVarSelect_MA_JOG_VELO"."$MA_JOG_VELO_Axis06_U2".token,
                                  Addr7 := "DB_NcVarSelect_MA_JOG_VELO_RAPID"."$MA_JOG_VELO_RAPID_Axis06_U2".token,
                                  Addr8 := "DB_NcVarSelect_M_MAX_AX_VELO"."$MA_JOG_VELO_Axis06_U2".token,
                                  Error => #sError,
                                  NDR => #sNDR,
                                  State => #sState,
                                  RD1 := #sAxis06_U2."$AA_IM",
                                  RD2 := #sAxis06_U2."$MA_POS_LIMIT_MINUS",
                                  RD3 := #sAxis06_U2."$MA_POS_LIMIT_MINUS2",
                                  RD4 := #sAxis06_U2."$MA_POS_LIMIT_PLUS",
                                  RD5 := #sAxis06_U2."$MA_POS_LIMIT_PLUS2",
                                  RD6 := #sAxis06_U2."$MA_JOG_VELO",
                                  RD7 := #sAxis06_U2."$MA_JOG_VELO_RAPID",
                                  RD8 := #sAxis06_U2."$MA_MAX_AX_VELO");
   END_REGION

   REGION Axis 07 V
       "LBP_ReadVar_DB_Axis07_V"(Req := NOT "Clock_10Hz",
                                 NumVar := 8,
                                 Addr1 := "DB_NcVarSelect_AA_IM"."$AA_IM_Axis07_V".token,
                                 Addr2 := "DB_NcVarSelect_MA_POS_LIMIT_MINUS"."$MA_POS_LIMIT_MINUS_Axis07_V".token,
                                 Addr3 := "DB_NcVarSelect_MA_POS_LIMIT_MINUS2"."$MA_POS_LIMIT_MINUS2_Axis07_V".token,
                                 Addr4 := "DB_NcVarSelect_MA_POS_LIMIT_PLUS"."$MA_POS_LIMIT_PLUS_Axis07_V".token,
                                 Addr5 := "DB_NcVarSelect_MA_POS_LIMIT_PLUS2"."$MA_POS_LIMIT_PLUS2_Axis07_V".token,
                                 Addr6 := "DB_NcVarSelect_MA_JOG_VELO"."$MA_JOG_VELO_Axis07_V".token,
                                 Addr7 := "DB_NcVarSelect_MA_JOG_VELO_RAPID"."$MA_JOG_VELO_RAPID_Axis07_V".token,
                                 Addr8 := "DB_NcVarSelect_M_MAX_AX_VELO"."$MA_JOG_VELO_Axis07_V".token,
                                 Error => #sError,
                                 NDR => #sNDR,
                                 State => #sState,
                                 RD1 := #sAxis07_V."$AA_IM",
                                 RD2 := #sAxis07_V."$MA_POS_LIMIT_MINUS",
                                 RD3 := #sAxis07_V."$MA_POS_LIMIT_MINUS2",
                                 RD4 := #sAxis07_V."$MA_POS_LIMIT_PLUS",
                                 RD5 := #sAxis07_V."$MA_POS_LIMIT_PLUS2",
                                 RD6 := #sAxis07_V."$MA_JOG_VELO",
                                 RD7 := #sAxis07_V."$MA_JOG_VELO_RAPID",
                                 RD8 := #sAxis07_V."$MA_MAX_AX_VELO");
   END_REGION

   REGION Axis 08 W
       "LBP_ReadVar_DB_Axis08_W"(Req := NOT "Clock_10Hz",
                                 NumVar := 8,
                                 Addr1 := "DB_NcVarSelect_AA_IM"."$AA_IM_Axis08_W".token,
                                 Addr2 := "DB_NcVarSelect_MA_POS_LIMIT_MINUS"."$MA_POS_LIMIT_MINUS_Axis08_W".token,
                                 Addr3 := "DB_NcVarSelect_MA_POS_LIMIT_MINUS2"."$MA_POS_LIMIT_MINUS2_Axis08_W".token,
                                 Addr4 := "DB_NcVarSelect_MA_POS_LIMIT_PLUS"."$MA_POS_LIMIT_PLUS_Axis08_W".token,
                                 Addr5 := "DB_NcVarSelect_MA_POS_LIMIT_PLUS2"."$MA_POS_LIMIT_PLUS2_Axis08_W".token,
                                 Addr6 := "DB_NcVarSelect_MA_JOG_VELO"."$MA_JOG_VELO_Axis08_W".token,
                                 Addr7 := "DB_NcVarSelect_MA_JOG_VELO_RAPID"."$MA_JOG_VELO_RAPID_Axis08_W".token,
                                 Addr8 := "DB_NcVarSelect_M_MAX_AX_VELO"."$MA_JOG_VELO_Axis08_W".token,
                                 Error => #sError,
                                 NDR => #sNDR,
                                 State => #sState,
                                 RD1 := #sAxis08_W."$AA_IM",
                                 RD2 := #sAxis08_W."$MA_POS_LIMIT_MINUS",
                                 RD3 := #sAxis08_W."$MA_POS_LIMIT_MINUS2",
                                 RD4 := #sAxis08_W."$MA_POS_LIMIT_PLUS",
                                 RD5 := #sAxis08_W."$MA_POS_LIMIT_PLUS2",
                                 RD6 := #sAxis08_W."$MA_JOG_VELO",
                                 RD7 := #sAxis08_W."$MA_JOG_VELO_RAPID",
                                 RD8 := #sAxis08_W."$MA_MAX_AX_VELO");
   END_REGION

   REGION Axis 09 ZL
       "LBP_ReadVar_DB_Axis09_ZL"(Req := "Clock_10Hz",
                                  NumVar := 8,
                                  Addr1 := "DB_NcVarSelect_AA_IM"."$AA_IM_Axis09_ZL".token,
                                  Addr2 := "DB_NcVarSelect_MA_POS_LIMIT_MINUS"."$MA_POS_LIMIT_MINUS_Axis09_ZL".token,
                                  Addr3 := "DB_NcVarSelect_MA_POS_LIMIT_MINUS2"."$MA_POS_LIMIT_MINUS2_Axis09_ZL".token,
                                  Addr4 := "DB_NcVarSelect_MA_POS_LIMIT_PLUS"."$MA_POS_LIMIT_PLUS_Axis09_ZL".token,
                                  Addr5 := "DB_NcVarSelect_MA_POS_LIMIT_PLUS2"."$MA_POS_LIMIT_PLUS2_Axis09_ZL".token,
                                  Addr6 := "DB_NcVarSelect_MA_JOG_VELO"."$MA_JOG_VELO_Axis09_ZL".token,
                                  Addr7 := "DB_NcVarSelect_MA_JOG_VELO_RAPID"."$MA_JOG_VELO_RAPID_Axis09_ZL".token,
                                  Addr8 := "DB_NcVarSelect_M_MAX_AX_VELO"."$MA_JOG_VELO_Axis09_ZL".token,
                                  Error => #sError,
                                  NDR => #sNDR,
                                  State => #sState,
                                  RD1 := #sAxis09_ZL."$AA_IM",
                                  RD2 := #sAxis09_ZL."$MA_POS_LIMIT_MINUS",
                                  RD3 := #sAxis09_ZL."$MA_POS_LIMIT_MINUS2",
                                  RD4 := #sAxis09_ZL."$MA_POS_LIMIT_PLUS",
                                  RD5 := #sAxis09_ZL."$MA_POS_LIMIT_PLUS2",
                                  RD6 := #sAxis09_ZL."$MA_JOG_VELO",
                                  RD7 := #sAxis09_ZL."$MA_JOG_VELO_RAPID",
                                  RD8 := #sAxis09_ZL."$MA_MAX_AX_VELO");
    END_REGION
END_FUNCTION_BLOCK

FUNCTION_BLOCK "FB_MCPManagement"   // FB421, SCL
{ S7_Optimized_Access := 'TRUE' }
// stored: AutoNumber false, MemoryReserve 100, SetENOAutomatically false
   VAR
      sRT_SingleBlock : R_TRIG;
      sSelectionAxe01Jog { S7_SetPoint := 'True'} : Bool;
      sSelectionAxe02Jog { S7_SetPoint := 'True'} : Bool;
      sSelectionAxe03Jog : Bool;
      sSelectionAxe04Jog : Bool;
      sSelectionAxe05Jog : Bool;
      sSelectionAxe06Jog : Bool;
      sSelectionAxe07Jog : Bool;
      sSelectionAxe08Jog : Bool;
      sSelectionAxe09Jog : Bool;
      sSelectionAxe10Jog : Bool;
      sSelectionAxe11Jog : Bool;
      sSelectionAxe12Jog : Bool;
      sSelectionAxe13Jog : Bool;
      sSelectionAxe14Jog : Bool;
      sSelectionAxe15Jog : Bool;
      sSelectionAxe16Jog : Bool;
      sSelectionAxe17Jog : Bool;
      sResetProgramEnmodeRef : Bool;
      sRT_McsWcs { S7_SetPoint := 'True'} : R_TRIG;
      sMemoFeedDisable { S7_SetPoint := 'True'} : Bool;
      sTONChanRef { S7_SetPoint := 'True'} : TON_TIME;
      sFP_TONChanRef { S7_SetPoint := 'True'} : R_TRIG;
   END_VAR
   VAR_TEMP
      tFeedrate : Byte;
      tStartTimerChanRef : Bool;
   END_VAR
BEGIN
   REGION Description header 
       //==================================================================================
       // POSALUX Swiss SA / (C) Copyright 2024
       //----------------------------------------------------------------------------------
       // Title: Management of the general MCP button functionalities
       // Comment/Function: 
       // Author: Gowsigan SRITHARAN
       // Engineering: TIA Portal v17
       //----------------------------------------------------------------------------------
       // Change log table:
       // Version  | Date     | Expert in charge | Changes applied
       // ---------|----------|------------------|------------------------------------
       // 00.00.01 | 20250411 | GSR              | First released version
       // 00.00.02 | 20251010 | WFA              | Femto 5a adaptation
       // ==================================================================================
   END_REGION

   REGION Call Mcp keyboard signals management
       "DB_McpKeyboardSignals"();
   END_REGION

   REGION General MCP buttons
       // JOG
       "LBP_ModeGroup".A_JOG := "MCP1_In".jog;
       "MCP1_Out".LEDjog := "LBP_ModeGroup".E_JOG;

       // MDA
       "LBP_ModeGroup".A_MDA := "MCP1_In".mda;
       "MCP1_Out".LEDmda := "LBP_ModeGroup".E_MDA;

       // AUTO
       "LBP_ModeGroup".A_AUTO := "MCP1_In".auto;
       "MCP1_Out".LEDauto := "LBP_ModeGroup".E_AUTO;

       // INC1
       "LBP_ModeGroup".A_INC1 := "MCP1_In".inc1 AND "LBP_ModeGroup".E_JOG;
       "MCP1_Out".LEDinc1 := "LBP_ModeGroup".E_INC1;

       // INC10
       "LBP_ModeGroup".A_INC10 := "MCP1_In".inc10 AND "LBP_ModeGroup".E_JOG;
       "MCP1_Out".LEDinc10 := "LBP_ModeGroup".E_INC10;

       // INC100
       "LBP_ModeGroup".A_INC100 := "MCP1_In".inc100 AND "LBP_ModeGroup".E_JOG;
       "MCP1_Out".LEDinc100 := "LBP_ModeGroup".E_INC100;

       // INC1000
       "LBP_ModeGroup".A_INC1000 := "MCP1_In".inc1000 AND "LBP_ModeGroup".E_JOG;
       "MCP1_Out".LEDinc1000 := "LBP_ModeGroup".E_INC1000;

       // INC10000
       "LBP_ModeGroup".A_INC10000 := "MCP1_In".inc10000 AND "LBP_ModeGroup".E_JOG;
       "MCP1_Out".LEDinc10000 := "LBP_ModeGroup".E_INC10000;

       // INCVAR
       "LBP_ModeGroup".A_INCVar := "MCP1_In".incVar AND "LBP_ModeGroup".E_JOG;
       "MCP1_Out".LEDincVar := "LBP_ModeGroup".E_INCVar;

       // RESET
       "LBP_Chan1".A_Reset := "MCP1_In".reset;

       // SINGLE BLOCK
       #sRT_SingleBlock(CLK := "MCP1_In".singleBlock);

       IF #sRT_SingleBlock.Q THEN
           "LBP_Chan1".A_SBL := NOT "LBP_Chan1".A_SBL;
       END_IF;

       "MCP1_Out".LEDsingleBlock := "LBP_Chan1".A_SBL;
   END_REGION

   REGION Selection axis in JOG

       // Mode JOG selection axe 01
       IF "MCP1_In".axisX AND "LBP_ModeGroup".E_JOG THEN
           #sSelectionAxe01Jog := TRUE;
           #sSelectionAxe02Jog := FALSE;
           #sSelectionAxe03Jog := FALSE;
           #sSelectionAxe04Jog := FALSE;
           #sSelectionAxe05Jog := FALSE;
           #sSelectionAxe06Jog := FALSE;
           #sSelectionAxe07Jog := FALSE;
           #sSelectionAxe08Jog := FALSE;
           #sSelectionAxe09Jog := FALSE;
       END_IF;

       // Mode JOG selection axe 02
       IF "MCP1_In".axisY AND "LBP_ModeGroup".E_JOG THEN
           #sSelectionAxe01Jog := FALSE;
           #sSelectionAxe02Jog := TRUE;
           #sSelectionAxe03Jog := FALSE;
           #sSelectionAxe04Jog := FALSE;
           #sSelectionAxe05Jog := FALSE;
           #sSelectionAxe06Jog := FALSE;
           #sSelectionAxe07Jog := FALSE;
           #sSelectionAxe08Jog := FALSE;
           #sSelectionAxe09Jog := FALSE;
       END_IF;

       // Mode JOG selection axe 03
       IF "MCP1_In".axisZ AND "LBP_ModeGroup".E_JOG THEN
           #sSelectionAxe01Jog := FALSE;
           #sSelectionAxe02Jog := FALSE;
           #sSelectionAxe03Jog := TRUE;
           #sSelectionAxe04Jog := FALSE;
           #sSelectionAxe05Jog := FALSE;
           #sSelectionAxe06Jog := FALSE;
           #sSelectionAxe07Jog := FALSE;
           #sSelectionAxe08Jog := FALSE;
           #sSelectionAxe09Jog := FALSE;
       END_IF;

       // Mode JOG selection axe 04
       IF "MCP1_In".axis4 AND "LBP_ModeGroup".E_JOG THEN
           #sSelectionAxe01Jog := FALSE;
           #sSelectionAxe02Jog := FALSE;
           #sSelectionAxe03Jog := FALSE;
           #sSelectionAxe04Jog := TRUE;
           #sSelectionAxe05Jog := FALSE;
           #sSelectionAxe06Jog := FALSE;
           #sSelectionAxe07Jog := FALSE;
           #sSelectionAxe08Jog := FALSE;
           #sSelectionAxe09Jog := FALSE;
       END_IF;

       // Mode JOG selection axe 05
       IF "MCP1_In".axis5 AND "LBP_ModeGroup".E_JOG THEN
           #sSelectionAxe01Jog := FALSE;
           #sSelectionAxe02Jog := FALSE;
           #sSelectionAxe03Jog := FALSE;
           #sSelectionAxe04Jog := FALSE;
           #sSelectionAxe05Jog := TRUE;
           #sSelectionAxe06Jog := FALSE;
           #sSelectionAxe07Jog := FALSE;
           #sSelectionAxe08Jog := FALSE;
           #sSelectionAxe09Jog := FALSE;
       END_IF;

       // Mode JOG selection axe 06
       IF "MCP1_In".axis6 AND "LBP_ModeGroup".E_JOG THEN
           #sSelectionAxe01Jog := FALSE;
           #sSelectionAxe02Jog := FALSE;
           #sSelectionAxe03Jog := FALSE;
           #sSelectionAxe04Jog := FALSE;
           #sSelectionAxe05Jog := FALSE;
           #sSelectionAxe06Jog := TRUE;
           #sSelectionAxe07Jog := FALSE;
           #sSelectionAxe08Jog := FALSE;
           #sSelectionAxe09Jog := FALSE;
       END_IF;

       // Mode JOG selection axe 07
       IF "MCP1_In".axis7 AND "LBP_ModeGroup".E_JOG THEN
           #sSelectionAxe01Jog := FALSE;
           #sSelectionAxe02Jog := FALSE;
           #sSelectionAxe03Jog := FALSE;
           #sSelectionAxe04Jog := FALSE;
           #sSelectionAxe05Jog := FALSE;
           #sSelectionAxe06Jog := FALSE;
           #sSelectionAxe07Jog := TRUE;
           #sSelectionAxe08Jog := FALSE;
           #sSelectionAxe09Jog := FALSE;
       END_IF;

       // Mode JOG selection axe 08
       IF "MCP1_In".axis8 AND "LBP_ModeGroup".E_JOG THEN
           #sSelectionAxe01Jog := FALSE;
           #sSelectionAxe02Jog := FALSE;
           #sSelectionAxe03Jog := FALSE;
           #sSelectionAxe04Jog := FALSE;
           #sSelectionAxe05Jog := FALSE;
           #sSelectionAxe06Jog := FALSE;
           #sSelectionAxe07Jog := FALSE;
           #sSelectionAxe08Jog := TRUE;
           #sSelectionAxe09Jog := FALSE;
       END_IF;

       // Mode JOG selection axe 09
       IF "MCP1_In".axis9 AND "LBP_ModeGroup".E_JOG THEN
           #sSelectionAxe01Jog := FALSE;
           #sSelectionAxe02Jog := FALSE;
           #sSelectionAxe03Jog := FALSE;
           #sSelectionAxe04Jog := FALSE;
           #sSelectionAxe05Jog := FALSE;
           #sSelectionAxe06Jog := FALSE;
           #sSelectionAxe07Jog := FALSE;
           #sSelectionAxe08Jog := FALSE;
           #sSelectionAxe09Jog := TRUE;
       END_IF;

       // Reset selection jog
       IF NOT "LBP_ModeGroup".E_JOG THEN
           #sSelectionAxe01Jog := FALSE;
           #sSelectionAxe02Jog := FALSE;
           #sSelectionAxe03Jog := FALSE;
           #sSelectionAxe04Jog := FALSE;
           #sSelectionAxe05Jog := FALSE;
           #sSelectionAxe06Jog := FALSE;
           #sSelectionAxe07Jog := FALSE;
           #sSelectionAxe08Jog := FALSE;
           #sSelectionAxe09Jog := FALSE;
       END_IF;

       // Led Axis
       "MCP1_Out".LEDaxisX := #sSelectionAxe01Jog;
       "MCP1_Out".LEDaxisY := #sSelectionAxe02Jog;
       "MCP1_Out".LEDaxisZ := #sSelectionAxe03Jog;
       "MCP1_Out".LEDaxis4 := #sSelectionAxe04Jog;
       "MCP1_Out".LEDaxis5 := #sSelectionAxe05Jog;
       "MCP1_Out".LEDaxis6 := #sSelectionAxe06Jog;
       "MCP1_Out".LEDaxis7 := #sSelectionAxe07Jog;
       "MCP1_Out".LEDaxis8 := #sSelectionAxe08Jog;
       "MCP1_Out".LEDaxis9 := #sSelectionAxe09Jog;
   END_REGION

   REGION Axis move in JOG
       // Axis 01
       IF #sSelectionAxe01Jog THEN
           "LBP_Axis01_X"."A_Plus" := "MCP1_In".plus;
           "LBP_Axis01_X".A_Minus := "MCP1_In".minus;
           "LBP_Axis01_X".A_RapidTrOR := "MCP1_In".rapidTraverse;
       END_IF;

       // Axis 02
       IF #sSelectionAxe02Jog THEN
           "LBP_Axis02_Y".A_Plus := "MCP1_In".plus;
           "LBP_Axis02_Y".A_Minus := "MCP1_In".minus;
           "LBP_Axis02_Y".A_RapidTrOR := "MCP1_In".rapidTraverse;
       END_IF;

       // Axis 03
       IF #sSelectionAxe03Jog THEN
           "LBP_Axis03_ZM".A_Plus := "MCP1_In".plus;
           "LBP_Axis03_ZM".A_Minus := "MCP1_In".minus;
           "LBP_Axis03_ZM".A_RapidTrOR := "MCP1_In".rapidTraverse;
       END_IF;

       // Axis 04
       IF #sSelectionAxe04Jog THEN
           "LBP_Axis04_B".A_Plus := "MCP1_In".plus;
           "LBP_Axis04_B".A_Minus := "MCP1_In".minus;
           "LBP_Axis04_B".A_RapidTrOR := "MCP1_In".rapidTraverse;
       END_IF;

       // Axis 05
       IF #sSelectionAxe05Jog THEN
           "LBP_Axis05_U1".A_Plus := "MCP1_In".plus;
           "LBP_Axis05_U1".A_Minus := "MCP1_In".minus;
           "LBP_Axis05_U1".A_RapidTrOR := "MCP1_In".rapidTraverse;
       END_IF;

       // Axis 06
       IF #sSelectionAxe06Jog THEN
           "LBP_Axis06_U2".A_Plus := "MCP1_In".plus;
           "LBP_Axis06_U2".A_Minus := "MCP1_In".minus;
           "LBP_Axis06_U2".A_RapidTrOR := "MCP1_In".rapidTraverse;
       END_IF;

       // Axe 07
       IF #sSelectionAxe07Jog THEN
           "LBP_Axis07_V".A_Plus := "MCP1_In".plus;
           "LBP_Axis07_V".A_Minus := "MCP1_In".minus;
           "LBP_Axis07_V".A_RapidTrOR := "MCP1_In".rapidTraverse;
       END_IF;

       // Axis 08
       IF #sSelectionAxe08Jog THEN
           "LBP_Axis08_W".A_Plus := "MCP1_In".plus;
           "LBP_Axis08_W".A_Minus := "MCP1_In".minus;
           "LBP_Axis08_W".A_RapidTrOR := "MCP1_In".rapidTraverse;
       END_IF;

       // Axis 09
       IF #sSelectionAxe09Jog THEN
           "LBP_Axis09_ZL".A_Plus := "MCP1_In".plus;
           "LBP_Axis09_ZL".A_Minus := "MCP1_In".minus;
           "LBP_Axis09_ZL".A_RapidTrOR := "MCP1_In".rapidTraverse;
       END_IF;
   END_REGION

   REGION Start and stop feedrate
   // FeedStart/Stop
   IF (NOT "MCP1_In".feedrateStop) AND (NOT "MCP1_In".feedrateStart) THEN
       #sMemoFeedDisable:= TRUE;
   ELSIF "MCP1_In".feedrateStop AND  "MCP1_In".feedrateStart THEN
       #sMemoFeedDisable:= FALSE;
   END_IF;
   "LBP_Chan1".A_FDdisable := #sMemoFeedDisable;

   // LED FeedStop
   "MCP1_Out".LEDfeedrateStop := #sMemoFeedDisable;
   "MCP1_Out".LEDfeedrateStart := NOT #sMemoFeedDisable;
   END_REGION

   REGION Channel feedrate override
       // Activation de la correction de l'avance
       "LBP_Chan1".A_FD_ORA := TRUE;

       #tFeedrate.%X0 := "MCP1_In".feedrateOvrA;
       #tFeedrate.%X1 := "MCP1_In".feedrateOvrB;
       #tFeedrate.%X2 := "MCP1_In".feedrateOvrC;
       #tFeedrate.%X3 := "MCP1_In".feedrateOvrD;
       #tFeedrate.%X4 := "MCP1_In".feedrateOvrE;
       #tFeedrate.%X5 := FALSE;
       #tFeedrate.%X6 := FALSE;
       #tFeedrate.%X7 := FALSE;

       // Forcing the override at 100% between 20% and 120% in manual/MDA mode WFA A REVOIR
       // IF NOT "LBP_ModeGroup".E_JOG AND #tFeedrate >= 8 THEN
       //     "LBP_Chan1".A_FD_OR := 26;
       // ELSE
           "LBP_Chan1".A_FD_OR     := #tFeedrate;
           "LBP_Axis01_X".A_FD_OR  := #tFeedrate;
           "LBP_Axis02_Y".A_FD_OR  := #tFeedrate;
           "LBP_Axis03_ZM".A_FD_OR := #tFeedrate;
           "LBP_Axis04_B".A_FD_OR  := #tFeedrate;
           "LBP_Axis05_U1".A_FD_OR := #tFeedrate;
           "LBP_Axis06_U2".A_FD_OR := #tFeedrate;
           "LBP_Axis07_V".A_FD_OR  := #tFeedrate;
           "LBP_Axis08_W".A_FD_OR  := #tFeedrate;
           "LBP_Axis09_ZL".A_FD_OR := #tFeedrate;
       // END_IF;
   END_REGION

   REGION Axis override
       // Allows modifying the movement speed OF the axis using the feed potentiometer
       "LBP_Axis01_X".A_ORactive  := TRUE;
       "LBP_Axis02_Y".A_ORactive  := TRUE;
       "LBP_Axis03_ZM".A_ORactive := TRUE;
       "LBP_Axis04_B".A_ORactive  := TRUE;
       "LBP_Axis05_U1".A_ORactive := TRUE;
       "LBP_Axis06_U2".A_ORactive := TRUE;
       "LBP_Axis07_V".A_ORactive  := TRUE;
       "LBP_Axis08_W".A_ORactive  := TRUE;
       "LBP_Axis09_ZL".A_ORactive := TRUE;
   END_REGION

   REGION Rapid traverse override active
       // Allows adjustment of the axis movement speed using the feed potentiometer
       "LBP_Chan1".A_RT_ORA := TRUE;
       "LBP_Chan1".A_RT_OR := "LBP_Chan1".A_FD_OR;
   END_REGION

   REGION Switching between MCS and WCS
       #sRT_McsWcs(CLK := "MCP1_In".mcsWcs OR  "LBP_HMI".E_ActWCS);
       IF #sRT_McsWcs.Q THEN
           "LBP_HMI".A_ActWCS := NOT "LBP_HMI".A_ActWCS;
       END_IF;
       "MCP1_Out".LEDmcsWcs := NOT "LBP_HMI".A_ActWCS;
   END_REGION

   REGION Key Switch signals
       "LBP_NC".A_Keyswitch0 := "MCP1_In".keySwitch0;
       "LBP_NC".A_Keyswitch1 := "MCP1_In".keySwitch1;
       "LBP_NC".A_Keyswitch2 := "MCP1_In".keySwitch2;
       "LBP_NC".A_Keyswitch3 := "MCP1_In".keySwitch3;
   END_REGION

   REGION Channel Referencing
       "LBP_ModeGroup".A_REF := "MCP1_In".refPoint;

       IF ("LBP_ModeGroup".E_REF
           AND NOT "LBP_Chan1".A_Ref)
           OR ("LBP_ModeGroup".E_REF
           AND "LBP_Chan1".A_Ref
           AND "Clock_1.25Hz") THEN
           "MCP1_Out".LEDrefPoint := TRUE;
       ELSE
           "MCP1_Out".LEDrefPoint := FALSE;
       END_IF;

       IF "LBP_ModeGroup".E_JOG
           AND "LBP_ModeGroup".E_REF
           AND "LBP_Chan1".A_NCStart THEN
           "LBP_Chan1".A_Ref := TRUE;
       END_IF;

       #tStartTimerChanRef :=
       "LBP_Chan1".E_AxesRef
       AND NOT "LBP_Chan1".E_Ref
       AND "LBP_Chan1".A_Ref
       AND "LBP_Chan1".E_ChanReset;

       #sTONChanRef(IN := #tStartTimerChanRef,
                    PT := T#500MS);

       #sFP_TONChanRef(CLK := #sTONChanRef.Q);

       IF #sFP_TONChanRef.Q THEN
           "LBP_ModeGroup".A_JOG := TRUE;
       END_IF;

       IF #sFP_TONChanRef.Q OR "LBP_Chan1".A_Reset THEN
           "LBP_Chan1".A_Ref := FALSE;
       END_IF;
   END_REGION

   REGION Reset group mode
       "LBP_ModeGroup".A_MGReset := "LBP_NC".E_NCKalarm AND "LBP_Chan1".A_Reset;
   END_REGION
END_FUNCTION_BLOCK

FUNCTION_BLOCK "FB_McpKeyboardSignals"   // FB420, SCL
{ S7_Optimized_Access := 'TRUE' }
// stored: AutoNumber false, MemoryReserve 100, SetENOAutomatically false
   VAR
      sK1_Powermeter : "FB_McpKeysSignals";
      sK2_GasAssist : "FB_McpKeysSignals";
      sK3_KeySaveParam : "FB_McpKeysSignals";
      sK4_GripperUndrilledPart : "FB_McpKeysSignals";
      sK5_GripperDrilledPart : "FB_McpKeysSignals";
      sK6_SITestStop : "FB_McpKeysSignals";
      sK7_FixtureClamp : "FB_McpKeysSignals";
      sK8_FixtureVacuum : "FB_McpKeysSignals";
      sK9_Aspiration : "FB_McpKeysSignals";
      sK10_LoaderAuto : "FB_McpKeysSignals";
      sK11_LoaderSemiAuto : "FB_McpKeysSignals";
      sK12_ObservationCamera : "FB_McpKeysSignals";
      sK13_MainDoor : "FB_McpKeysSignals";
      sK14_WarmUp : "FB_McpKeysSignals";
      sK15_MachineLight : "FB_McpKeysSignals";
      sStartCycle { S7_SetPoint := 'True'} : "FB_McpKeysSignals";
      sAlarmReset { S7_SetPoint := 'True'} : "FB_McpKeysSignals";
      sPowerOFF { S7_SetPoint := 'True'} : "FB_McpKeysSignals";
      sShutdownPC { S7_SetPoint := 'True'} : "FB_McpKeysSignals";
      sLightTest { S7_SetPoint := 'True'} : "FB_McpKeysSignals";
      sPowerON { S7_SetPoint := 'True'} : "FB_McpKeysSignals";
      sRemoteOpenShutter { S7_SetPoint := 'True'} : "FB_McpKeysSignals";
      sAx10_LaserArea { S7_SetPoint := 'True'} : "FB_McpKeysSignals";
      sAx11_ChannelSelection { S7_SetPoint := 'True'} : "FB_McpKeysSignals";
   END_VAR
   VAR_TEMP
      tNoLed : Bool;   // Index for loop
   END_VAR
BEGIN
   REGION Description header 
       //==================================================================================
       // POSALUX Swiss SA / (C) Copyright 2024
       //----------------------------------------------------------------------------------
       // Title: Management of inputs and outputs for MCP buttons
       // Comment/Function: 
       //
       // Author: Gowsigan SRITHARAN
       // Engineering: TIA Portal v17
       //----------------------------------------------------------------------------------
       // Change log table:
       // Version  | Date     | Expert in charge | Changes applied
       // ---------|----------|------------------|------------------------------------
       // 00.00.01 | 20241120 | GSR              | First released version
       // 00.00.02 | 20250911 | WFA              | PB - LED Management with multi-instance FB
       // ==================================================================================
   END_REGION

   REGION Customer keys (Middle panel)
       // Key1 : Powermeter
       #sK1_Powermeter(iKeyHWStatus := "MCP1_In".customerKey1,
                       oLedHWStatus =>"MCP1_Out".LEDcustomerKey1);

       // Key2 : Gas Assist
       #sK2_GasAssist(iKeyHWStatus := "MCP1_In".customerKey2,
                      oLedHWStatus => "MCP1_Out".LEDcustomerKey2);

       // Key3 : Save Param
       #sK3_KeySaveParam(iKeyHWStatus := "MCP1_In".customerKey3,
                         oLedHWStatus => "MCP1_Out".LEDcustomerKey3);

       // Key4 : Gripper Undrilled Part
       #sK4_GripperUndrilledPart(iKeyHWStatus := "MCP1_In".customerKey4,
                                 oLedHWStatus => "MCP1_Out".LEDcustomerKey4);

       // Key5 : Gripper Drilled Part
       #sK5_GripperDrilledPart(iKeyHWStatus := "MCP1_In".customerKey5,
                               oLedHWStatus => "MCP1_Out".LEDcustomerKey5);

       // Key6 : SI Test Stop
       #sK6_SITestStop(iKeyHWStatus := "MCP1_In".customerKey6,
                       oLedHWStatus => "MCP1_Out".LEDcustomerKey6);

       // Key7 : Fixture Clamp
       #sK7_FixtureClamp(iKeyHWStatus := "MCP1_In".customerKey7,
                         oLedHWStatus => "MCP1_Out".LEDcustomerKey7);

       // Key8 : Fixture Vacuum
       #sK8_FixtureVacuum(iKeyHWStatus := "MCP1_In".customerKey8,
                          oLedHWStatus => "MCP1_Out".LEDcustomerKey8);

       // Key9 : Aspiration
       #sK9_Aspiration(iKeyHWStatus := "MCP1_In".customerKey9,
                       oLedHWStatus => "MCP1_Out".LEDcustomerKey9);

       // Key10 : Loader Mode Auto
       #sK10_LoaderAuto(iKeyHWStatus := "MCP1_In".customerKey10,
                        oLedHWStatus => "MCP1_Out".LEDcustomerKey10);

       // Key11 : Loader Mode Semi Auto
       #sK11_LoaderSemiAuto(iKeyHWStatus := "MCP1_In".customerKey11,
                            oLedHWStatus => "MCP1_Out".LEDcustomerKey11);

       // Key12 : Observation Camera
       #sK12_ObservationCamera(iKeyHWStatus := "MCP1_In".customerKey12,
                               oLedHWStatus => "MCP1_Out".LEDcustomerKey12);

       // Key13 : Main Door
       #sK13_MainDoor(iKeyHWStatus := "MCP1_In".customerKey13,
                      oLedHWStatus => "MCP1_Out".LEDcustomerKey13);

       // Key14 : Warm Up
       #sK14_WarmUp(iKeyHWStatus := "MCP1_In".customerKey14,
                    oLedHWStatus => "MCP1_Out".LEDcustomerKey14);

       // Key15 : Camera Light
       #sK15_MachineLight(iKeyHWStatus := "MCP1_In".customerKey15,
                          oLedHWStatus => "MCP1_Out".LEDcustomerKey15);
   END_REGION Customer keys    

